LIN {X 0.113,Y -541.801,Z 1483.606,A 0.000,B 0.000,C 90.000,E1 144.975} C_DIS
LIN {X 0.190,Y -543.941,Z 1483.601,A 0.000,B 0.000,C 90.000,E1 144.116} C_DIS
LIN {X -0.031,Y -545.794,Z 1483.596,A 0.000,B 0.000,C 90.000,E1 143.290} C_DIS
LIN {X 0.087,Y -547.494,Z 1483.591,A 0.000,B 0.000,C 90.000,E1 142.431} C_DIS
LIN {X -0.159,Y -549.493,Z 1483.585,A 0.000,B 0.000,C 90.000,E1 141.331} C_DIS
LIN {X -0.082,Y -550.826,Z 1483.580,A 0.000,B 0.000,C 90.000,E1 140.481} C_DIS
LIN {X -0.278,Y -552.385,Z 1483.574,A 0.000,B 0.000,C 90.000,E1 139.380} C_DIS
LIN {X -0.042,Y -554.152,Z 1483.566,A 0.000,B 0.000,C 90.000,E1 137.957} C_DIS
LIN {X 0.124,Y -555.386,Z 1483.560,A 0.000,B 0.000,C 90.000,E1 136.824} C_DIS
LIN {X -0.011,Y -556.776,Z 1483.552,A 0.000,B 0.000,C 90.000,E1 135.445} C_DIS
LIN {X -0.192,Y -557.702,Z 1483.546,A 0.000,B 0.000,C 90.000,E1 134.352} C_DIS
LIN {X -0.236,Y -558.934,Z 1483.537,A 0.000,B 0.000,C 90.000,E1 132.690} C_DIS
LIN {X 0.038,Y -559.548,Z 1483.531,A 0.000,B 0.000,C 90.000,E1 131.553} C_DIS
LIN {X -0.100,Y -559.973,Z 1483.525,A 0.000,B 0.000,C 90.000,E1 130.458} C_DIS
LIN {X -0.079,Y -560.380,Z 1483.517,A 0.000,B 0.000,C 90.000,E1 129.072} C_DIS
LIN {X -0.139,Y -560.620,Z 1483.511,A 0.000,B 0.000,C 90.000,E1 127.971} C_DIS
LIN {X 0.086,Y -560.790,Z 1483.500,A 0.000,B 0.000,C 90.000,E1 126.011} C_DIS
LIN {X 0.236,Y -560.719,Z 1483.492,A 0.000,B 0.000,C 90.000,E1 124.612} C_DIS
LIN {X 0.120,Y -560.448,Z 1483.479,A 0.000,B 0.000,C 90.000,E1 122.133} C_DIS
LIN {X -0.123,Y -560.638,Z 1483.465,A 0.000,B 0.000,C 90.000,E1 119.667} C_DIS
LIN {X -0.105,Y -560.801,Z 1483.457,A 0.000,B 0.000,C 90.000,E1 118.281} C_DIS
LIN {X -0.254,Y -561.104,Z 1483.446,A 0.000,B 0.000,C 90.000,E1 116.360} C_DIS
LIN {X 0.113,Y -561.555,Z 1483.436,A 0.000,B 0.000,C 90.000,E1 114.387} C_DIS
LIN {X -0.087,Y -561.949,Z 1483.428,A 0.000,B 0.000,C 90.000,E1 113.025} C_DIS
LIN {X 0.050,Y -562.381,Z 1483.419,A 0.000,B 0.000,C 90.000,E1 111.354} C_DIS
LIN {X -0.136,Y -562.769,Z 1483.411,A 0.000,B 0.000,C 90.000,E1 109.993} C_DIS
LIN {X 0.014,Y -563.133,Z 1483.403,A 0.000,B 0.000,C 90.000,E1 108.598} C_DIS
LIN {X 0.310,Y -563.530,Z 1483.394,A 0.000,B 0.000,C 90.000,E1 106.913} C_DIS
LIN {X 0.145,Y -563.929,Z 1483.386,A 0.000,B 0.000,C 90.000,E1 105.552} C_DIS
LIN {X -0.090,Y -564.549,Z 1483.376,A 0.000,B 0.000,C 90.000,E1 103.647} C_DIS
LIN {X 0.020,Y -565.015,Z 1483.370,A 0.000,B 0.000,C 90.000,E1 102.535} C_DIS
LIN {X -0.077,Y -565.623,Z 1483.360,A 0.000,B 0.000,C 90.000,E1 100.894} C_DIS
LIN {X -0.271,Y -566.373,Z 1483.351,A 0.000,B 0.000,C 90.000,E1 99.265} C_DIS
LIN {X 0.194,Y -567.231,Z 1483.341,A 0.000,B 0.000,C 90.000,E1 97.296} C_DIS
LIN {X 0.039,Y -568.297,Z 1483.330,A 0.000,B 0.000,C 90.000,E1 95.391} C_DIS
LIN {X -0.192,Y -569.521,Z 1483.319,A 0.000,B 0.000,C 90.000,E1 93.498} C_DIS
LIN {X -0.100,Y -570.416,Z 1483.312,A 0.000,B 0.000,C 90.000,E1 92.121} C_DIS
LIN {X 0.139,Y -571.623,Z 1483.303,A 0.000,B 0.000,C 90.000,E1 90.458} C_DIS
LIN {X 0.096,Y -573.230,Z 1483.291,A 0.000,B 0.000,C 90.000,E1 88.282} C_DIS
LIN {X -0.156,Y -574.365,Z 1483.281,A 0.000,B 0.000,C 90.000,E1 86.674} C_DIS
LIN {X -0.233,Y -575.774,Z 1483.271,A 0.000,B 0.000,C 90.000,E1 84.780} C_DIS
LIN {X 0.197,Y -577.016,Z 1483.262,A 0.000,B 0.000,C 90.000,E1 83.109} C_DIS
LIN {X 0.153,Y -578.302,Z 1483.253,A 0.000,B 0.000,C 90.000,E1 81.489} C_DIS
LIN {X 0.232,Y -579.653,Z 1483.244,A 0.000,B 0.000,C 90.000,E1 79.859} C_DIS
LIN {X -0.230,Y -580.999,Z 1483.235,A 0.000,B 0.000,C 90.000,E1 78.285} C_DIS
LIN {X 0.122,Y -581.962,Z 1483.229,A 0.000,B 0.000,C 90.000,E1 77.173} C_DIS
LIN {X -0.044,Y -583.179,Z 1483.220,A 0.000,B 0.000,C 90.000,E1 75.574} C_DIS
LIN {X 0.148,Y -584.105,Z 1483.212,A 0.000,B 0.000,C 90.000,E1 74.212} C_DIS
LIN {X -0.217,Y -584.893,Z 1483.205,A 0.000,B 0.000,C 90.000,E1 72.906} C_DIS
LIN {X 0.005,Y -585.755,Z 1483.196,A 0.000,B 0.000,C 90.000,E1 71.275} C_DIS
LIN {X 0.027,Y -586.436,Z 1483.189,A 0.000,B 0.000,C 90.000,E1 69.934} C_DIS
LIN {X 0.060,Y -587.171,Z 1483.181,A 0.000,B 0.000,C 90.000,E1 68.592} C_DIS
LIN {X 0.159,Y -588.653,Z 1483.168,A 0.000,B 0.000,C 90.000,E1 66.177} C_DIS
LIN {X -0.177,Y -589.158,Z 1483.163,A 0.000,B 0.000,C 90.000,E1 65.409} C_DIS
LIN {X 0.136,Y -590.165,Z 1483.153,A 0.000,B 0.000,C 90.000,E1 63.512} C_DIS
LIN {X 0.102,Y -591.682,Z 1483.141,A 0.000,B 0.000,C 90.000,E1 61.385} C_DIS
LIN {X 0.071,Y -592.910,Z 1483.132,A 0.000,B 0.000,C 90.000,E1 59.793} C_DIS
LIN {X -0.038,Y -594.394,Z 1483.122,A 0.000,B 0.000,C 90.000,E1 57.946} C_DIS
LIN {X -0.325,Y -595.276,Z 1483.116,A 0.000,B 0.000,C 90.000,E1 56.914} C_DIS
LIN {X -0.143,Y -596.583,Z 1483.107,A 0.000,B 0.000,C 90.000,E1 55.308} C_DIS
LIN {X 0.069,Y -597.764,Z 1483.098,A 0.000,B 0.000,C 90.000,E1 53.703} C_DIS
LIN {X -0.063,Y -598.634,Z 1483.091,A 0.000,B 0.000,C 90.000,E1 52.396} C_DIS
LIN {X -0.178,Y -599.244,Z 1483.084,A 0.000,B 0.000,C 90.000,E1 51.090} C_DIS
LIN {X 0.094,Y -599.916,Z 1483.076,A 0.000,B 0.000,C 90.000,E1 49.747} C_DIS
LIN {X 0.114,Y -600.179,Z 1483.073,A 0.000,B 0.000,C 90.000,E1 49.218} C_DIS
LIN {X 0.158,Y -600.394,Z 1483.068,A 0.000,B 0.000,C 90.000,E1 48.162} C_DIS
LIN {X -0.017,Y -600.455,Z 1483.060,A 0.000,B 0.000,C 90.000,E1 46.863} C_DIS
LIN {X 0.202,Y -600.413,Z 1483.056,A 0.000,B 0.000,C 90.000,E1 46.053} C_DIS
LIN {X 0.007,Y -600.117,Z 1483.049,A 0.000,B 0.000,C 90.000,E1 44.757} C_DIS
LIN {X 0.225,Y -599.782,Z 1483.044,A 0.000,B 0.000,C 90.000,E1 43.947} C_DIS
LIN {X -0.401,Y -598.890,Z 1483.037,A 0.000,B 0.000,C 90.000,E1 42.690} C_DIS
LIN {X 0.246,Y -597.651,Z 1483.030,A 0.000,B 0.000,C 90.000,E1 41.310} C_DIS
LIN {X 0.254,Y -596.494,Z 1483.024,A 0.000,B 0.000,C 90.000,E1 40.253} C_DIS
LIN {X 0.019,Y -595.474,Z 1483.019,A 0.000,B 0.000,C 90.000,E1 39.483} C_DIS
LIN {X -0.165,Y -593.500,Z 1483.012,A 0.000,B 0.000,C 90.000,E1 38.177} C_DIS
LIN {X 0.096,Y -591.141,Z 1483.005,A 0.000,B 0.000,C 90.000,E1 36.824} C_DIS
LIN {X -0.365,Y -588.888,Z 1482.999,A 0.000,B 0.000,C 90.000,E1 35.804} C_DIS
LIN {X -0.101,Y -586.984,Z 1482.994,A 0.000,B 0.000,C 90.000,E1 34.978} C_DIS
LIN {X -0.339,Y -584.811,Z 1482.990,A 0.000,B 0.000,C 90.000,E1 34.199} C_DIS
LIN {X 0.028,Y -583.207,Z 1482.987,A 0.000,B 0.000,C 90.000,E1 33.627} C_DIS
LIN {X 0.058,Y -581.442,Z 1482.984,A 0.000,B 0.000,C 90.000,E1 33.086} C_DIS
LIN {X 0.084,Y -577.555,Z 1482.978,A 0.000,B 0.000,C 90.000,E1 32.005} C_DIS
LIN {X 0.078,Y -575.345,Z 1482.975,A 0.000,B 0.000,C 90.000,E1 31.465} C_DIS
LIN {X -0.110,Y -571.657,Z 1482.970,A 0.000,B 0.000,C 90.000,E1 30.669} C_DIS
LIN {X -0.249,Y -568.337,Z 1482.967,A 0.000,B 0.000,C 90.000,E1 30.001} C_DIS
LIN {X -0.111,Y -563.299,Z 1482.961,A 0.000,B 0.000,C 90.000,E1 29.027} C_DIS
LIN {X 0.167,Y -559.372,Z 1482.957,A 0.000,B 0.000,C 90.000,E1 28.309} C_DIS
LIN {X -0.086,Y -554.990,Z 1482.954,A 0.000,B 0.000,C 90.000,E1 27.641} C_DIS
LIN {X 0.081,Y -551.973,Z 1482.951,A 0.000,B 0.000,C 90.000,E1 27.206} C_DIS
LIN {X -0.007,Y -548.380,Z 1482.949,A 0.000,B 0.000,C 90.000,E1 26.796} C_DIS
LIN {X 0.252,Y -545.487,Z 1482.947,A 0.000,B 0.000,C 90.000,E1 26.488} C_DIS
LIN {X 0.255,Y -543.930,Z 1482.947,A 0.000,B 0.000,C 90.000,E1 26.360} C_DIS
LIN {X -0.225,Y -541.263,Z 1482.946,A 0.000,B 0.000,C 90.000,E1 26.232} C_DIS
LIN {X 0.063,Y -538.976,Z 1482.945,A 0.000,B 0.000,C 90.000,E1 26.104} C_DIS
LIN {X -0.136,Y -537.794,Z 1482.945,A 0.000,B 0.000,C 90.000,E1 26.104} C_DIS
LIN {X -0.121,Y -384.370,Z 1482.945,A 0.000,B 0.000,C 90.000,E1 26.104} C_DIS
LIN {X 0.078,Y -383.033,Z 1482.939,A 0.000,B 0.000,C 90.000,E1 24.951} C_DIS
LIN {X -0.114,Y -381.912,Z 1482.935,A 0.000,B 0.000,C 90.000,E1 24.259} C_DIS
LIN {X 0.134,Y -375.526,Z 1482.909,A 0.000,B 0.000,C 90.000,E1 19.504} C_DIS
LIN {X 0.003,Y -373.426,Z 1482.896,A 0.000,B 0.000,C 90.000,E1 17.330} C_DIS
LIN {X 0.014,Y -367.903,Z 1482.868,A 0.000,B 0.000,C 90.000,E1 12.175} C_DIS
LIN {X -0.043,Y -366.502,Z 1482.855,A 0.000,B 0.000,C 90.000,E1 9.962} C_DIS
LIN {X -0.108,Y -361.802,Z 1482.822,A 0.000,B 0.000,C 90.000,E1 4.012} C_DIS
LIN {X 0.138,Y -360.903,Z 1482.801,A 0.000,B 0.000,C 90.000,E1 0.229} C_DIS
LIN {X -0.053,Y -359.426,Z 1482.770,A 0.000,B 0.000,C 90.000,E1 354.546} C_DIS
LIN {X 0.070,Y -358.890,Z 1482.759,A 0.000,B 0.000,C 90.000,E1 352.648} C_DIS
LIN {X -0.020,Y -359.563,Z 1482.726,A 0.000,B 0.000,C 90.000,E1 346.645} C_DIS
LIN {X 0.001,Y -361.801,Z 1482.684,A 0.000,B 0.000,C 90.000,E1 339.135} C_DIS
LIN {X -0.154,Y -362.053,Z 1482.680,A 0.000,B 0.000,C 90.000,E1 338.411} C_DIS
LIN {X 0.189,Y -365.980,Z 1482.643,A 0.000,B 0.000,C 90.000,E1 331.641} C_DIS
LIN {X 0.029,Y -366.387,Z 1482.639,A 0.000,B 0.000,C 90.000,E1 330.923} C_DIS
LIN {X -0.031,Y -371.355,Z 1482.604,A 0.000,B 0.000,C 90.000,E1 324.642} C_DIS
LIN {X -0.043,Y -371.766,Z 1482.602,A 0.000,B 0.000,C 90.000,E1 324.276} C_DIS
LIN {X 0.013,Y -377.358,Z 1482.567,A 0.000,B 0.000,C 90.000,E1 318.038} C_DIS
LIN {X 0.012,Y -378.235,Z 1482.563,A 0.000,B 0.000,C 90.000,E1 317.310} C_DIS
LIN {X 0.002,Y -383.940,Z 1482.531,A 0.000,B 0.000,C 90.000,E1 311.515} C_DIS
LIN {X 0.088,Y -384.893,Z 1482.527,A 0.000,B 0.000,C 90.000,E1 310.782} C_DIS
LIN {X 0.262,Y -390.610,Z 1482.495,A 0.000,B 0.000,C 90.000,E1 305.025} C_DIS
LIN {X 0.106,Y -391.104,Z 1482.493,A 0.000,B 0.000,C 90.000,E1 304.692} C_DIS
LIN {X 0.022,Y -391.648,Z 1482.489,A 0.000,B 0.000,C 90.000,E1 303.992} C_DIS
LIN {X -0.080,Y -396.825,Z 1482.459,A 0.000,B 0.000,C 90.000,E1 298.693} C_DIS
LIN {X -0.210,Y -397.120,Z 1482.457,A 0.000,B 0.000,C 90.000,E1 298.359} C_DIS
LIN {X -0.055,Y -401.597,Z 1482.426,A 0.000,B 0.000,C 90.000,E1 292.717} C_DIS
LIN {X 0.222,Y -404.659,Z 1482.395,A 0.000,B 0.000,C 90.000,E1 287.094} C_DIS
LIN {X -0.079,Y -404.735,Z 1482.391,A 0.000,B 0.000,C 90.000,E1 286.441} C_DIS
LIN {X 0.214,Y -406.099,Z 1482.364,A 0.000,B 0.000,C 90.000,E1 281.535} C_DIS
LIN {X -0.176,Y -406.094,Z 1482.362,A 0.000,B 0.000,C 90.000,E1 281.243} C_DIS
LIN {X -0.097,Y -405.680,Z 1482.333,A 0.000,B 0.000,C 90.000,E1 276.024} C_DIS
LIN {X -0.165,Y -405.058,Z 1482.328,A 0.000,B 0.000,C 90.000,E1 274.992} C_DIS
LIN {X -0.060,Y -403.497,Z 1482.304,A 0.000,B 0.000,C 90.000,E1 270.802} C_DIS
LIN {X -0.092,Y -403.288,Z 1482.302,A 0.000,B 0.000,C 90.000,E1 270.458} C_DIS
LIN {X 0.091,Y -398.931,Z 1482.271,A 0.000,B 0.000,C 90.000,E1 264.837} C_DIS
LIN {X -0.040,Y -393.108,Z 1482.242,A 0.000,B 0.000,C 90.000,E1 259.567} C_DIS
LIN {X -0.079,Y -392.835,Z 1482.240,A 0.000,B 0.000,C 90.000,E1 259.218} C_DIS
LIN {X 0.034,Y -385.993,Z 1482.212,A 0.000,B 0.000,C 90.000,E1 254.212} C_DIS
LIN {X -0.026,Y -385.267,Z 1482.208,A 0.000,B 0.000,C 90.000,E1 253.504} C_DIS
LIN {X -0.004,Y -384.768,Z 1482.206,A 0.000,B 0.000,C 90.000,E1 253.142} C_DIS
LIN {X 0.221,Y -377.973,Z 1482.182,A 0.000,B 0.000,C 90.000,E1 248.773} C_DIS
LIN {X -0.044,Y -376.233,Z 1482.174,A 0.000,B 0.000,C 90.000,E1 247.358} C_DIS
LIN {X 0.057,Y -374.944,Z 1482.170,A 0.000,B 0.000,C 90.000,E1 246.613} C_DIS
LIN {X -0.208,Y -368.417,Z 1482.148,A 0.000,B 0.000,C 90.000,E1 242.615} C_DIS
LIN {X 0.097,Y -366.047,Z 1482.137,A 0.000,B 0.000,C 90.000,E1 240.717} C_DIS
LIN {X 0.004,Y -359.196,Z 1482.115,A 0.000,B 0.000,C 90.000,E1 236.628} C_DIS
LIN {X 0.021,Y -355.842,Z 1482.100,A 0.000,B 0.000,C 90.000,E1 233.989} C_DIS
LIN {X -0.173,Y -348.793,Z 1482.075,A 0.000,B 0.000,C 90.000,E1 229.461} C_DIS
LIN {X -0.097,Y -346.185,Z 1482.062,A 0.000,B 0.000,C 90.000,E1 227.148} C_DIS
LIN {X -0.088,Y -345.065,Z 1482.058,A 0.000,B 0.000,C 90.000,E1 226.377} C_DIS
LIN {X 0.094,Y -338.586,Z 1482.030,A 0.000,B 0.000,C 90.000,E1 221.310} C_DIS
LIN {X 0.094,Y -336.840,Z 1482.019,A 0.000,B 0.000,C 90.000,E1 219.358} C_DIS
LIN {X 0.014,Y -330.861,Z 1481.988,A 0.000,B 0.000,C 90.000,E1 213.865} C_DIS
LIN {X 0.149,Y -329.296,Z 1481.975,A 0.000,B 0.000,C 90.000,E1 211.465} C_DIS
LIN {X -0.154,Y -324.669,Z 1481.942,A 0.000,B 0.000,C 90.000,E1 205.540} C_DIS
LIN {X 0.174,Y -323.837,Z 1481.928,A 0.000,B 0.000,C 90.000,E1 203.078} C_DIS
LIN {X -0.017,Y -321.124,Z 1481.881,A 0.000,B 0.000,C 90.000,E1 194.662} C_DIS
LIN {X 0.138,Y -320.932,Z 1481.877,A 0.000,B 0.000,C 90.000,E1 193.828} C_DIS
LIN {X -0.076,Y -321.562,Z 1481.832,A 0.000,B 0.000,C 90.000,E1 185.796} C_DIS
LIN {X -0.143,Y -324.415,Z 1481.790,A 0.000,B 0.000,C 90.000,E1 178.165} C_DIS
LIN {X -0.141,Y -325.376,Z 1481.783,A 0.000,B 0.000,C 90.000,E1 176.963} C_DIS
LIN {X -0.100,Y -329.112,Z 1481.750,A 0.000,B 0.000,C 90.000,E1 170.971} C_DIS
LIN {X 0.061,Y -334.260,Z 1481.726,A 0.000,B 0.000,C 90.000,E1 166.589} C_DIS
LIN {X 0.067,Y -335.488,Z 1481.719,A 0.000,B 0.000,C 90.000,E1 165.408} C_DIS
LIN {X 0.143,Y -340.932,Z 1481.695,A 0.000,B 0.000,C 90.000,E1 161.094} C_DIS
LIN {X -0.172,Y -342.138,Z 1481.691,A 0.000,B 0.000,C 90.000,E1 160.369} C_DIS
LIN {X -0.058,Y -347.939,Z 1481.667,A 0.000,B 0.000,C 90.000,E1 156.102} C_DIS
LIN {X 0.037,Y -354.622,Z 1481.647,A 0.000,B 0.000,C 90.000,E1 152.436} C_DIS
LIN {X 0.000,Y -354.671,Z 1481.647,A 0.000,B 0.000,C 90.000,E1 152.410} C_DIS
LIN {X -0.047,Y -501.646,Z 1481.647,A 0.000,B 0.000,C 90.000,E1 152.410} C_DIS
LIN {X -0.075,Y -505.220,Z 1481.646,A 0.000,B 0.000,C 90.000,E1 152.281} C_DIS
LIN {X -0.137,Y -507.377,Z 1481.645,A 0.000,B 0.000,C 90.000,E1 152.153} C_DIS
LIN {X -0.108,Y -509.939,Z 1481.644,A 0.000,B 0.000,C 90.000,E1 151.948} C_DIS
LIN {X -0.018,Y -513.664,Z 1481.642,A 0.000,B 0.000,C 90.000,E1 151.563} C_DIS
LIN {X 0.194,Y -515.980,Z 1481.641,A 0.000,B 0.000,C 90.000,E1 151.257} C_DIS
LIN {X -0.069,Y -519.084,Z 1481.638,A 0.000,B 0.000,C 90.000,E1 150.845} C_DIS
LIN {X -0.026,Y -522.481,Z 1481.635,A 0.000,B 0.000,C 90.000,E1 150.255} C_DIS
LIN {X -0.117,Y -526.265,Z 1481.631,A 0.000,B 0.000,C 90.000,E1 149.537} C_DIS
LIN {X 0.091,Y -529.473,Z 1481.627,A 0.000,B 0.000,C 90.000,E1 148.791} C_DIS
LIN {X 0.207,Y -531.888,Z 1481.624,A 0.000,B 0.000,C 90.000,E1 148.201} C_DIS
LIN {X -0.117,Y -534.035,Z 1481.620,A 0.000,B 0.000,C 90.000,E1 147.661} C_DIS
LIN {X 0.013,Y -536.921,Z 1481.615,A 0.000,B 0.000,C 90.000,E1 146.786} C_DIS
LIN {X 0.026,Y -539.502,Z 1481.611,A 0.000,B 0.000,C 90.000,E1 145.928} C_DIS
LIN {X -0.232,Y -541.972,Z 1481.606,A 0.000,B 0.000,C 90.000,E1 145.102} C_DIS
LIN {X 0.289,Y -544.154,Z 1481.601,A 0.000,B 0.000,C 90.000,E1 144.196} C_DIS
LIN {X 0.069,Y -546.018,Z 1481.597,A 0.000,B 0.000,C 90.000,E1 143.371} C_DIS
LIN {X -0.201,Y -548.230,Z 1481.590,A 0.000,B 0.000,C 90.000,E1 142.271} C_DIS
LIN {X -0.056,Y -549.722,Z 1481.586,A 0.000,B 0.000,C 90.000,E1 141.412} C_DIS
LIN {X 0.078,Y -551.419,Z 1481.579,A 0.000,B 0.000,C 90.000,E1 140.275} C_DIS
LIN {X -0.116,Y -552.960,Z 1481.573,A 0.000,B 0.000,C 90.000,E1 139.175} C_DIS
LIN {X 0.067,Y -554.326,Z 1481.567,A 0.000,B 0.000,C 90.000,E1 138.038} C_DIS
LIN {X -0.111,Y -555.828,Z 1481.559,A 0.000,B 0.000,C 90.000,E1 136.662} C_DIS
LIN {X 0.152,Y -557.194,Z 1481.552,A 0.000,B 0.000,C 90.000,E1 135.243} C_DIS
LIN {X 0.035,Y -558.250,Z 1481.544,A 0.000,B 0.000,C 90.000,E1 133.866} C_DIS
LIN {X -0.041,Y -559.241,Z 1481.536,A 0.000,B 0.000,C 90.000,E1 132.486} C_DIS
LIN {X -0.176,Y -559.800,Z 1481.530,A 0.000,B 0.000,C 90.000,E1 131.391} C_DIS
LIN {X -0.226,Y -560.240,Z 1481.522,A 0.000,B 0.000,C 90.000,E1 130.011} C_DIS
LIN {X -0.199,Y -560.596,Z 1481.515,A 0.000,B 0.000,C 90.000,E1 128.624} C_DIS
LIN {X -0.163,Y -560.744,Z 1481.507,A 0.000,B 0.000,C 90.000,E1 127.237} C_DIS
LIN {X 0.318,Y -560.835,Z 1481.499,A 0.000,B 0.000,C 90.000,E1 125.804} C_DIS
LIN {X -0.084,Y -560.757,Z 1481.493,A 0.000,B 0.000,C 90.000,E1 124.739} C_DIS
LIN {X 0.057,Y -560.447,Z 1481.478,A 0.000,B 0.000,C 90.000,E1 121.957} C_DIS
LIN {X 0.033,Y -560.619,Z 1481.465,A 0.000,B 0.000,C 90.000,E1 119.745} C_DIS
LIN {X -0.146,Y -560.817,Z 1481.456,A 0.000,B 0.000,C 90.000,E1 118.103} C_DIS
LIN {X -0.086,Y -561.090,Z 1481.447,A 0.000,B 0.000,C 90.000,E1 116.437} C_DIS
LIN {X -0.221,Y -561.538,Z 1481.436,A 0.000,B 0.000,C 90.000,E1 114.515} C_DIS
LIN {X 0.116,Y -562.010,Z 1481.427,A 0.000,B 0.000,C 90.000,E1 112.823} C_DIS
LIN {X 0.038,Y -562.486,Z 1481.418,A 0.000,B 0.000,C 90.000,E1 111.173} C_DIS
LIN {X -0.145,Y -562.844,Z 1481.410,A 0.000,B 0.000,C 90.000,E1 109.812} C_DIS
LIN {X 0.147,Y -563.278,Z 1481.401,A 0.000,B 0.000,C 90.000,E1 108.127} C_DIS
LIN {X 0.064,Y -563.801,Z 1481.390,A 0.000,B 0.000,C 90.000,E1 106.205} C_DIS
LIN {X 0.215,Y -564.288,Z 1481.381,A 0.000,B 0.000,C 90.000,E1 104.537} C_DIS
LIN {X -0.156,Y -565.017,Z 1481.370,A 0.000,B 0.000,C 90.000,E1 102.647} C_DIS
LIN {X 0.296,Y -565.653,Z 1481.361,A 0.000,B 0.000,C 90.000,E1 100.950} C_DIS
LIN {X -0.207,Y -566.629,Z 1481.349,A 0.000,B 0.000,C 90.000,E1 98.803} C_DIS
LIN {X -0.196,Y -567.682,Z 1481.337,A 0.000,B 0.000,C 90.000,E1 96.606} C_DIS
LIN {X 0.066,Y -568.632,Z 1481.328,A 0.000,B 0.000,C 90.000,E1 94.935} C_DIS
LIN {X -0.114,Y -569.903,Z 1481.317,A 0.000,B 0.000,C 90.000,E1 93.037} C_DIS
LIN {X 0.107,Y -571.045,Z 1481.308,A 0.000,B 0.000,C 90.000,E1 91.375} C_DIS
LIN {X 0.208,Y -572.009,Z 1481.300,A 0.000,B 0.000,C 90.000,E1 90.000} C_DIS
LIN {X -0.106,Y -573.258,Z 1481.291,A 0.000,B 0.000,C 90.000,E1 88.396} C_DIS
LIN {X 0.217,Y -574.426,Z 1481.282,A 0.000,B 0.000,C 90.000,E1 86.731} C_DIS
LIN {X 0.144,Y -575.851,Z 1481.271,A 0.000,B 0.000,C 90.000,E1 84.837} C_DIS
LIN {X 0.005,Y -577.111,Z 1481.262,A 0.000,B 0.000,C 90.000,E1 83.223} C_DIS
LIN {X -0.247,Y -578.199,Z 1481.255,A 0.000,B 0.000,C 90.000,E1 81.894} C_DIS
LIN {X -0.270,Y -579.539,Z 1481.246,A 0.000,B 0.000,C 90.000,E1 80.274} C_DIS
LIN {X -0.061,Y -580.925,Z 1481.237,A 0.000,B 0.000,C 90.000,E1 78.634} C_DIS
LIN {X 0.190,Y -582.338,Z 1481.228,A 0.000,B 0.000,C 90.000,E1 76.992} C_DIS
LIN {X -0.110,Y -583.542,Z 1481.219,A 0.000,B 0.000,C 90.000,E1 75.408} C_DIS
LIN {X 0.076,Y -584.419,Z 1481.211,A 0.000,B 0.000,C 90.000,E1 74.047} C_DIS
LIN {X -0.121,Y -585.200,Z 1481.204,A 0.000,B 0.000,C 90.000,E1 72.725} C_DIS
LIN {X -0.225,Y -586.253,Z 1481.194,A 0.000,B 0.000,C 90.000,E1 70.859} C_DIS
LIN {X -0.249,Y -587.353,Z 1481.182,A 0.000,B 0.000,C 90.000,E1 68.720} C_DIS
LIN {X 0.315,Y -588.454,Z 1481.171,A 0.000,B 0.000,C 90.000,E1 66.794} C_DIS
LIN {X 0.050,Y -589.326,Z 1481.164,A 0.000,B 0.000,C 90.000,E1 65.485} C_DIS
LIN {X -0.170,Y -590.341,Z 1481.154,A 0.000,B 0.000,C 90.000,E1 63.640} C_DIS
LIN {X -0.096,Y -591.604,Z 1481.143,A 0.000,B 0.000,C 90.000,E1 61.769} C_DIS
LIN {X -0.319,Y -592.662,Z 1481.136,A 0.000,B 0.000,C 90.000,E1 60.461} C_DIS
LIN {X -0.224,Y -594.346,Z 1481.124,A 0.000,B 0.000,C 90.000,E1 58.329} C_DIS
LIN {X -0.111,Y -595.444,Z 1481.117,A 0.000,B 0.000,C 90.000,E1 56.993} C_DIS
LIN {X 0.070,Y -596.770,Z 1481.108,A 0.000,B 0.000,C 90.000,E1 55.388} C_DIS
LIN {X -0.200,Y -597.960,Z 1481.099,A 0.000,B 0.000,C 90.000,E1 53.829} C_DIS
LIN {X 0.151,Y -598.865,Z 1481.092,A 0.000,B 0.000,C 90.000,E1 52.477} C_DIS
LIN {X 0.038,Y -599.514,Z 1481.084,A 0.000,B 0.000,C 90.000,E1 51.170} C_DIS
LIN {X 0.312,Y -600.176,Z 1481.077,A 0.000,B 0.000,C 90.000,E1 49.828} C_DIS
LIN {X 0.119,Y -600.525,Z 1481.073,A 0.000,B 0.000,C 90.000,E1 49.057} C_DIS
LIN {X 0.381,Y -600.692,Z 1481.068,A 0.000,B 0.000,C 90.000,E1 48.243} C_DIS
LIN {X -0.228,Y -600.762,Z 1481.061,A 0.000,B 0.000,C 90.000,E1 46.986} C_DIS
LIN {X -0.001,Y -600.734,Z 1481.057,A 0.000,B 0.000,C 90.000,E1 46.176} C_DIS
LIN {X 0.241,Y -600.466,Z 1481.049,A 0.000,B 0.000,C 90.000,E1 44.838} C_DIS
LIN {X 0.254,Y -599.989,Z 1481.043,A 0.000,B 0.000,C 90.000,E1 43.785} C_DIS
LIN {X 0.072,Y -599.083,Z 1481.036,A 0.000,B 0.000,C 90.000,E1 42.486} C_DIS
LIN {X 0.051,Y -598.104,Z 1481.030,A 0.000,B 0.000,C 90.000,E1 41.434} C_DIS
LIN {X 0.059,Y -596.947,Z 1481.024,A 0.000,B 0.000,C 90.000,E1 40.378} C_DIS
LIN {X 0.050,Y -595.527,Z 1481.019,A 0.000,B 0.000,C 90.000,E1 39.322} C_DIS
LIN {X 0.110,Y -593.991,Z 1481.013,A 0.000,B 0.000,C 90.000,E1 38.257} C_DIS
LIN {X -0.093,Y -591.687,Z 1481.005,A 0.000,B 0.000,C 90.000,E1 36.950} C_DIS
LIN {X -0.073,Y -589.493,Z 1480.999,A 0.000,B 0.000,C 90.000,E1 35.884} C_DIS
LIN {X -0.283,Y -587.620,Z 1480.995,A 0.000,B 0.000,C 90.000,E1 35.105} C_DIS
LIN {X -0.030,Y -585.505,Z 1480.990,A 0.000,B 0.000,C 90.000,E1 34.278} C_DIS
LIN {X -0.286,Y -583.094,Z 1480.986,A 0.000,B 0.000,C 90.000,E1 33.499} C_DIS
LIN {X -0.234,Y -579.480,Z 1480.980,A 0.000,B 0.000,C 90.000,E1 32.418} C_DIS
LIN {X -0.225,Y -577.441,Z 1480.977,A 0.000,B 0.000,C 90.000,E1 31.878} C_DIS
LIN {X -0.090,Y -573.965,Z 1480.973,A 0.000,B 0.000,C 90.000,E1 31.052} C_DIS
LIN {X 0.114,Y -569.519,Z 1480.967,A 0.000,B 0.000,C 90.000,E1 30.079} C_DIS
LIN {X -0.141,Y -563.024,Z 1480.960,A 0.000,B 0.000,C 90.000,E1 28.871} C_DIS
LIN {X -0.035,Y -559.907,Z 1480.957,A 0.000,B 0.000,C 90.000,E1 28.309} C_DIS
LIN {X 0.209,Y -555.559,Z 1480.953,A 0.000,B 0.000,C 90.000,E1 27.590} C_DIS
LIN {X 0.030,Y -551.830,Z 1480.950,A 0.000,B 0.000,C 90.000,E1 27.052} C_DIS
LIN {X 0.182,Y -548.690,Z 1480.948,A 0.000,B 0.000,C 90.000,E1 26.616} C_DIS
LIN {X -0.173,Y -544.957,Z 1480.946,A 0.000,B 0.000,C 90.000,E1 26.232} C_DIS
LIN {X 0.146,Y -542.086,Z 1480.944,A 0.000,B 0.000,C 90.000,E1 25.924} C_DIS
LIN {X 0.096,Y -540.475,Z 1480.943,A 0.000,B 0.000,C 90.000,E1 25.796} C_DIS
LIN {X 0.170,Y -538.760,Z 1480.943,A 0.000,B 0.000,C 90.000,E1 25.668} C_DIS
LIN {X 0.035,Y -535.864,Z 1480.942,A 0.000,B 0.000,C 90.000,E1 25.540} C_DIS
LIN {X -0.035,Y -534.505,Z 1480.942,A 0.000,B 0.000,C 90.000,E1 25.515} C_DIS
LIN {X -0.054,Y -383.662,Z 1480.942,A 0.000,B 0.000,C 90.000,E1 25.515} C_DIS
LIN {X 0.191,Y -382.637,Z 1480.937,A 0.000,B 0.000,C 90.000,E1 24.643} C_DIS
LIN {X 0.130,Y -375.997,Z 1480.911,A 0.000,B 0.000,C 90.000,E1 19.939} C_DIS
LIN {X -0.006,Y -373.524,Z 1480.897,A 0.000,B 0.000,C 90.000,E1 17.402} C_DIS
LIN {X 0.033,Y -367.958,Z 1480.868,A 0.000,B 0.000,C 90.000,E1 12.243} C_DIS
LIN {X 0.051,Y -366.538,Z 1480.856,A 0.000,B 0.000,C 90.000,E1 10.018} C_DIS
LIN {X -0.020,Y -365.428,Z 1480.850,A 0.000,B 0.000,C 90.000,E1 8.916} C_DIS
LIN {X -0.055,Y -361.273,Z 1480.814,A 0.000,B 0.000,C 90.000,E1 2.579} C_DIS
LIN {X -0.130,Y -360.906,Z 1480.802,A 0.000,B 0.000,C 90.000,E1 0.344} C_DIS
LIN {X 0.044,Y -359.764,Z 1480.786,A 0.000,B 0.000,C 90.000,E1 357.535} C_DIS
LIN {X -0.053,Y -359.426,Z 1480.770,A 0.000,B 0.000,C 90.000,E1 354.546} C_DIS
LIN {X 0.070,Y -358.890,Z 1480.759,A 0.000,B 0.000,C 90.000,E1 352.648} C_DIS
LIN {X -0.020,Y -359.563,Z 1480.726,A 0.000,B 0.000,C 90.000,E1 346.645} C_DIS
LIN {X 0.001,Y -361.801,Z 1480.684,A 0.000,B 0.000,C 90.000,E1 339.135} C_DIS
LIN {X -0.154,Y -362.053,Z 1480.680,A 0.000,B 0.000,C 90.000,E1 338.411} C_DIS
LIN {X 0.189,Y -365.980,Z 1480.643,A 0.000,B 0.000,C 90.000,E1 331.641} C_DIS
LIN {X 0.029,Y -366.387,Z 1480.639,A 0.000,B 0.000,C 90.000,E1 330.923} C_DIS
LIN {X -0.031,Y -371.355,Z 1480.604,A 0.000,B 0.000,C 90.000,E1 324.642} C_DIS
LIN {X -0.043,Y -371.766,Z 1480.602,A 0.000,B 0.000,C 90.000,E1 324.276} C_DIS
LIN {X 0.013,Y -377.358,Z 1480.567,A 0.000,B 0.000,C 90.000,E1 318.038} C_DIS
LIN {X 0.012,Y -378.235,Z 1480.563,A 0.000,B 0.000,C 90.000,E1 317.310} C_DIS
LIN {X 0.002,Y -383.940,Z 1480.531,A 0.000,B 0.000,C 90.000,E1 311.515} C_DIS
LIN {X 0.088,Y -384.893,Z 1480.527,A 0.000,B 0.000,C 90.000,E1 310.782} C_DIS
LIN {X 0.262,Y -390.610,Z 1480.495,A 0.000,B 0.000,C 90.000,E1 305.025} C_DIS
LIN {X 0.106,Y -391.104,Z 1480.493,A 0.000,B 0.000,C 90.000,E1 304.692} C_DIS
LIN {X 0.022,Y -391.648,Z 1480.489,A 0.000,B 0.000,C 90.000,E1 303.992} C_DIS
LIN {X -0.080,Y -396.825,Z 1480.459,A 0.000,B 0.000,C 90.000,E1 298.693} C_DIS
LIN {X -0.210,Y -397.120,Z 1480.457,A 0.000,B 0.000,C 90.000,E1 298.359} C_DIS
LIN {X -0.055,Y -401.597,Z 1480.426,A 0.000,B 0.000,C 90.000,E1 292.717} C_DIS
LIN {X 0.222,Y -404.659,Z 1480.395,A 0.000,B 0.000,C 90.000,E1 287.094} C_DIS
LIN {X -0.079,Y -404.735,Z 1480.391,A 0.000,B 0.000,C 90.000,E1 286.441} C_DIS
LIN {X 0.214,Y -406.099,Z 1480.364,A 0.000,B 0.000,C 90.000,E1 281.535} C_DIS
LIN {X -0.176,Y -406.094,Z 1480.362,A 0.000,B 0.000,C 90.000,E1 281.243} C_DIS
LIN {X -0.097,Y -405.680,Z 1480.333,A 0.000,B 0.000,C 90.000,E1 276.024} C_DIS
LIN {X -0.165,Y -405.058,Z 1480.328,A 0.000,B 0.000,C 90.000,E1 274.992} C_DIS
LIN {X -0.060,Y -403.497,Z 1480.304,A 0.000,B 0.000,C 90.000,E1 270.802} C_DIS
LIN {X -0.092,Y -403.288,Z 1480.302,A 0.000,B 0.000,C 90.000,E1 270.458} C_DIS
LIN {X 0.091,Y -398.931,Z 1480.271,A 0.000,B 0.000,C 90.000,E1 264.837} C_DIS
LIN {X -0.040,Y -393.108,Z 1480.242,A 0.000,B 0.000,C 90.000,E1 259.567} C_DIS
LIN {X -0.079,Y -392.835,Z 1480.240,A 0.000,B 0.000,C 90.000,E1 259.218} C_DIS
LIN {X 0.034,Y -385.993,Z 1480.212,A 0.000,B 0.000,C 90.000,E1 254.212} C_DIS
LIN {X -0.026,Y -385.267,Z 1480.208,A 0.000,B 0.000,C 90.000,E1 253.504} C_DIS
LIN {X -0.004,Y -384.768,Z 1480.206,A 0.000,B 0.000,C 90.000,E1 253.142} C_DIS
LIN {X 0.221,Y -377.973,Z 1480.182,A 0.000,B 0.000,C 90.000,E1 248.773} C_DIS
LIN {X -0.044,Y -376.233,Z 1480.174,A 0.000,B 0.000,C 90.000,E1 247.358} C_DIS
LIN {X 0.057,Y -374.944,Z 1480.170,A 0.000,B 0.000,C 90.000,E1 246.613} C_DIS
LIN {X -0.208,Y -368.417,Z 1480.148,A 0.000,B 0.000,C 90.000,E1 242.615} C_DIS
LIN {X 0.097,Y -366.047,Z 1480.137,A 0.000,B 0.000,C 90.000,E1 240.717} C_DIS
LIN {X 0.004,Y -359.196,Z 1480.115,A 0.000,B 0.000,C 90.000,E1 236.628} C_DIS
LIN {X 0.021,Y -355.842,Z 1480.100,A 0.000,B 0.000,C 90.000,E1 233.989} C_DIS
LIN {X -0.173,Y -348.793,Z 1480.075,A 0.000,B 0.000,C 90.000,E1 229.461} C_DIS
LIN {X -0.097,Y -346.185,Z 1480.062,A 0.000,B 0.000,C 90.000,E1 227.148} C_DIS
LIN {X -0.088,Y -345.065,Z 1480.058,A 0.000,B 0.000,C 90.000,E1 226.377} C_DIS
LIN {X 0.094,Y -338.586,Z 1480.030,A 0.000,B 0.000,C 90.000,E1 221.310} C_DIS
LIN {X 0.094,Y -336.840,Z 1480.019,A 0.000,B 0.000,C 90.000,E1 219.358} C_DIS
LIN {X 0.014,Y -330.861,Z 1479.988,A 0.000,B 0.000,C 90.000,E1 213.865} C_DIS
LIN {X 0.149,Y -329.296,Z 1479.975,A 0.000,B 0.000,C 90.000,E1 211.465} C_DIS
LIN {X -0.154,Y -324.669,Z 1479.942,A 0.000,B 0.000,C 90.000,E1 205.540} C_DIS
LIN {X 0.174,Y -323.837,Z 1479.928,A 0.000,B 0.000,C 90.000,E1 203.078} C_DIS
LIN {X -0.017,Y -321.124,Z 1479.881,A 0.000,B 0.000,C 90.000,E1 194.662} C_DIS
LIN {X 0.138,Y -320.932,Z 1479.877,A 0.000,B 0.000,C 90.000,E1 193.828} C_DIS
LIN {X -0.076,Y -321.562,Z 1479.832,A 0.000,B 0.000,C 90.000,E1 185.796} C_DIS
LIN {X -0.143,Y -324.415,Z 1479.790,A 0.000,B 0.000,C 90.000,E1 178.165} C_DIS
LIN {X -0.141,Y -325.376,Z 1479.783,A 0.000,B 0.000,C 90.000,E1 176.963} C_DIS
LIN {X -0.100,Y -329.112,Z 1479.750,A 0.000,B 0.000,C 90.000,E1 170.971} C_DIS
LIN {X 0.061,Y -334.260,Z 1479.726,A 0.000,B 0.000,C 90.000,E1 166.589} C_DIS
LIN {X 0.067,Y -335.488,Z 1479.719,A 0.000,B 0.000,C 90.000,E1 165.408} C_DIS
LIN {X 0.143,Y -340.932,Z 1479.695,A 0.000,B 0.000,C 90.000,E1 161.094} C_DIS
LIN {X -0.172,Y -342.138,Z 1479.691,A 0.000,B 0.000,C 90.000,E1 160.369} C_DIS
LIN {X -0.058,Y -347.939,Z 1479.667,A 0.000,B 0.000,C 90.000,E1 156.102} C_DIS
LIN {X -0.069,Y -353.576,Z 1479.650,A 0.000,B 0.000,C 90.000,E1 152.999} C_DIS
LIN {X -0.123,Y -497.290,Z 1479.650,A 0.000,B 0.000,C 90.000,E1 152.999} C_DIS
LIN {X -0.140,Y -500.027,Z 1479.650,A 0.000,B 0.000,C 90.000,E1 152.922} C_DIS
LIN {X 0.062,Y -501.637,Z 1479.649,A 0.000,B 0.000,C 90.000,E1 152.820} C_DIS
LIN {X -0.116,Y -504.385,Z 1479.648,A 0.000,B 0.000,C 90.000,E1 152.666} C_DIS
LIN {X 0.104,Y -506.939,Z 1479.647,A 0.000,B 0.000,C 90.000,E1 152.436} C_DIS
LIN {X -0.279,Y -510.846,Z 1479.645,A 0.000,B 0.000,C 90.000,E1 152.103} C_DIS
LIN {X -0.007,Y -514.398,Z 1479.642,A 0.000,B 0.000,C 90.000,E1 151.641} C_DIS
LIN {X 0.094,Y -516.525,Z 1479.641,A 0.000,B 0.000,C 90.000,E1 151.335} C_DIS
LIN {X 0.114,Y -520.206,Z 1479.638,A 0.000,B 0.000,C 90.000,E1 150.745} C_DIS
LIN {X 0.261,Y -524.228,Z 1479.634,A 0.000,B 0.000,C 90.000,E1 149.999} C_DIS
LIN {X 0.045,Y -526.497,Z 1479.631,A 0.000,B 0.000,C 90.000,E1 149.587} C_DIS
LIN {X -0.168,Y -530.315,Z 1479.626,A 0.000,B 0.000,C 90.000,E1 148.742} C_DIS
LIN {X 0.231,Y -532.670,Z 1479.623,A 0.000,B 0.000,C 90.000,E1 148.122} C_DIS
LIN {X -0.087,Y -534.770,Z 1479.620,A 0.000,B 0.000,C 90.000,E1 147.582} C_DIS
LIN {X 0.054,Y -537.604,Z 1479.615,A 0.000,B 0.000,C 90.000,E1 146.707} C_DIS
LIN {X 0.063,Y -539.360,Z 1479.612,A 0.000,B 0.000,C 90.000,E1 146.135} C_DIS
LIN {X 0.272,Y -542.614,Z 1479.606,A 0.000,B 0.000,C 90.000,E1 144.975} C_DIS
LIN {X 0.039,Y -544.727,Z 1479.601,A 0.000,B 0.000,C 90.000,E1 144.149} C_DIS
LIN {X 0.107,Y -546.008,Z 1479.598,A 0.000,B 0.000,C 90.000,E1 143.577} C_DIS
LIN {X -0.161,Y -548.199,Z 1479.592,A 0.000,B 0.000,C 90.000,E1 142.477} C_DIS
LIN {X 0.037,Y -550.182,Z 1479.585,A 0.000,B 0.000,C 90.000,E1 141.331} C_DIS
LIN {X 0.180,Y -551.843,Z 1479.579,A 0.000,B 0.000,C 90.000,E1 140.194} C_DIS
LIN {X -0.006,Y -553.357,Z 1479.573,A 0.000,B 0.000,C 90.000,E1 139.094} C_DIS
LIN {X 0.124,Y -554.376,Z 1479.568,A 0.000,B 0.000,C 90.000,E1 138.243} C_DIS
LIN {X -0.023,Y -555.909,Z 1479.560,A 0.000,B 0.000,C 90.000,E1 136.863} C_DIS
LIN {X -0.166,Y -557.207,Z 1479.553,A 0.000,B 0.000,C 90.000,E1 135.486} C_DIS
LIN {X -0.281,Y -558.302,Z 1479.545,A 0.000,B 0.000,C 90.000,E1 134.109} C_DIS
LIN {X 0.022,Y -559.320,Z 1479.537,A 0.000,B 0.000,C 90.000,E1 132.690} C_DIS
LIN {X -0.117,Y -559.880,Z 1479.531,A 0.000,B 0.000,C 90.000,E1 131.595} C_DIS
LIN {X 0.169,Y -560.250,Z 1479.525,A 0.000,B 0.000,C 90.000,E1 130.458} C_DIS
LIN {X -0.148,Y -560.614,Z 1479.516,A 0.000,B 0.000,C 90.000,E1 128.830} C_DIS
LIN {X -0.116,Y -560.784,Z 1479.508,A 0.000,B 0.000,C 90.000,E1 127.443} C_DIS
LIN {X 0.364,Y -560.894,Z 1479.500,A 0.000,B 0.000,C 90.000,E1 126.011} C_DIS
LIN {X -0.038,Y -560.803,Z 1479.494,A 0.000,B 0.000,C 90.000,E1 124.945} C_DIS
LIN {X -0.157,Y -560.458,Z 1479.480,A 0.000,B 0.000,C 90.000,E1 122.467} C_DIS
LIN {X -0.196,Y -560.559,Z 1479.468,A 0.000,B 0.000,C 90.000,E1 120.256} C_DIS
LIN {X -0.091,Y -560.791,Z 1479.457,A 0.000,B 0.000,C 90.000,E1 118.309} C_DIS
LIN {X 0.226,Y -561.062,Z 1479.448,A 0.000,B 0.000,C 90.000,E1 116.616} C_DIS
LIN {X -0.152,Y -561.466,Z 1479.437,A 0.000,B 0.000,C 90.000,E1 114.719} C_DIS
LIN {X 0.194,Y -562.002,Z 1479.428,A 0.000,B 0.000,C 90.000,E1 113.025} C_DIS
LIN {X 0.125,Y -562.562,Z 1479.417,A 0.000,B 0.000,C 90.000,E1 111.099} C_DIS
LIN {X -0.336,Y -563.053,Z 1479.407,A 0.000,B 0.000,C 90.000,E1 109.214} C_DIS
LIN {X -0.177,Y -563.396,Z 1479.399,A 0.000,B 0.000,C 90.000,E1 107.819} C_DIS
LIN {X 0.276,Y -563.935,Z 1479.388,A 0.000,B 0.000,C 90.000,E1 105.843} C_DIS
LIN {X 0.038,Y -564.559,Z 1479.378,A 0.000,B 0.000,C 90.000,E1 103.939} C_DIS
LIN {X 0.093,Y -565.307,Z 1479.367,A 0.000,B 0.000,C 90.000,E1 102.007} C_DIS
LIN {X -0.170,Y -565.847,Z 1479.359,A 0.000,B 0.000,C 90.000,E1 100.658} C_DIS
LIN {X -0.281,Y -566.720,Z 1479.349,A 0.000,B 0.000,C 90.000,E1 98.746} C_DIS
LIN {X -0.201,Y -567.782,Z 1479.336,A 0.000,B 0.000,C 90.000,E1 96.543} C_DIS
LIN {X 0.000,Y -568.739,Z 1479.327,A 0.000,B 0.000,C 90.000,E1 94.878} C_DIS
LIN {X -0.176,Y -570.010,Z 1479.317,A 0.000,B 0.000,C 90.000,E1 92.980} C_DIS
LIN {X 0.048,Y -571.185,Z 1479.307,A 0.000,B 0.000,C 90.000,E1 91.318} C_DIS
LIN {X -0.282,Y -572.345,Z 1479.298,A 0.000,B 0.000,C 90.000,E1 89.714} C_DIS
LIN {X -0.160,Y -573.408,Z 1479.291,A 0.000,B 0.000,C 90.000,E1 88.339} C_DIS
LIN {X 0.166,Y -574.607,Z 1479.282,A 0.000,B 0.000,C 90.000,E1 86.674} C_DIS
LIN {X 0.095,Y -576.042,Z 1479.271,A 0.000,B 0.000,C 90.000,E1 84.780} C_DIS
LIN {X -0.040,Y -577.320,Z 1479.262,A 0.000,B 0.000,C 90.000,E1 83.166} C_DIS
LIN {X -0.291,Y -578.441,Z 1479.255,A 0.000,B 0.000,C 90.000,E1 81.837} C_DIS
LIN {X 0.136,Y -579.561,Z 1479.247,A 0.000,B 0.000,C 90.000,E1 80.443} C_DIS
LIN {X -0.101,Y -581.190,Z 1479.237,A 0.000,B 0.000,C 90.000,E1 78.578} C_DIS
LIN {X 0.153,Y -582.612,Z 1479.228,A 0.000,B 0.000,C 90.000,E1 76.937} C_DIS
LIN {X 0.186,Y -583.644,Z 1479.220,A 0.000,B 0.000,C 90.000,E1 75.589} C_DIS
LIN {X -0.189,Y -584.519,Z 1479.213,A 0.000,B 0.000,C 90.000,E1 74.283} C_DIS
LIN {X -0.155,Y -585.446,Z 1479.204,A 0.000,B 0.000,C 90.000,E1 72.670} C_DIS
LIN {X -0.067,Y -586.524,Z 1479.193,A 0.000,B 0.000,C 90.000,E1 70.786} C_DIS
LIN {X 0.055,Y -587.461,Z 1479.183,A 0.000,B 0.000,C 90.000,E1 68.901} C_DIS
LIN {X -0.262,Y -588.717,Z 1479.171,A 0.000,B 0.000,C 90.000,E1 66.794} C_DIS
LIN {X 0.259,Y -589.560,Z 1479.164,A 0.000,B 0.000,C 90.000,E1 65.409} C_DIS
LIN {X -0.050,Y -590.756,Z 1479.152,A 0.000,B 0.000,C 90.000,E1 63.307} C_DIS
LIN {X -0.036,Y -591.667,Z 1479.144,A 0.000,B 0.000,C 90.000,E1 61.975} C_DIS
LIN {X -0.070,Y -592.934,Z 1479.135,A 0.000,B 0.000,C 90.000,E1 60.383} C_DIS
LIN {X 0.040,Y -594.641,Z 1479.124,A 0.000,B 0.000,C 90.000,E1 58.250} C_DIS
LIN {X 0.164,Y -595.725,Z 1479.116,A 0.000,B 0.000,C 90.000,E1 56.914} C_DIS
LIN {X 0.017,Y -597.075,Z 1479.108,A 0.000,B 0.000,C 90.000,E1 55.341} C_DIS
LIN {X -0.257,Y -598.256,Z 1479.099,A 0.000,B 0.000,C 90.000,E1 53.783} C_DIS
LIN {X 0.090,Y -599.187,Z 1479.091,A 0.000,B 0.000,C 90.000,E1 52.431} C_DIS
LIN {X 0.351,Y -599.855,Z 1479.084,A 0.000,B 0.000,C 90.000,E1 51.090} C_DIS
LIN {X -0.213,Y -600.500,Z 1479.077,A 0.000,B 0.000,C 90.000,E1 49.828} C_DIS
LIN {X 0.051,Y -600.835,Z 1479.072,A 0.000,B 0.000,C 90.000,E1 49.013} C_DIS
LIN {X -0.137,Y -600.995,Z 1479.068,A 0.000,B 0.000,C 90.000,E1 48.243} C_DIS
LIN {X 0.108,Y -601.059,Z 1479.061,A 0.000,B 0.000,C 90.000,E1 46.905} C_DIS
LIN {X -0.078,Y -601.019,Z 1479.056,A 0.000,B 0.000,C 90.000,E1 46.134} C_DIS
LIN {X -0.264,Y -600.763,Z 1479.049,A 0.000,B 0.000,C 90.000,E1 44.838} C_DIS
LIN {X -0.247,Y -600.272,Z 1479.043,A 0.000,B 0.000,C 90.000,E1 43.785} C_DIS
LIN {X -0.019,Y -599.355,Z 1479.036,A 0.000,B 0.000,C 90.000,E1 42.447} C_DIS
LIN {X -0.222,Y -598.668,Z 1479.031,A 0.000,B 0.000,C 90.000,E1 41.676} C_DIS
LIN {X -0.202,Y -597.524,Z 1479.026,A 0.000,B 0.000,C 90.000,E1 40.620} C_DIS
LIN {X -0.199,Y -596.162,Z 1479.020,A 0.000,B 0.000,C 90.000,E1 39.564} C_DIS
LIN {X 0.001,Y -594.246,Z 1479.012,A 0.000,B 0.000,C 90.000,E1 38.222} C_DIS
LIN {X 0.266,Y -591.951,Z 1479.005,A 0.000,B 0.000,C 90.000,E1 36.870} C_DIS
LIN {X 0.286,Y -589.750,Z 1478.999,A 0.000,B 0.000,C 90.000,E1 35.804} C_DIS
LIN {X 0.075,Y -587.883,Z 1478.995,A 0.000,B 0.000,C 90.000,E1 35.025} C_DIS
LIN {X -0.157,Y -585.776,Z 1478.990,A 0.000,B 0.000,C 90.000,E1 34.246} C_DIS
LIN {X 0.069,Y -583.363,Z 1478.986,A 0.000,B 0.000,C 90.000,E1 33.420} C_DIS
LIN {X 0.120,Y -579.782,Z 1478.980,A 0.000,B 0.000,C 90.000,E1 32.339} C_DIS
LIN {X 0.129,Y -577.744,Z 1478.977,A 0.000,B 0.000,C 90.000,E1 31.799} C_DIS
LIN {X -0.034,Y -574.284,Z 1478.972,A 0.000,B 0.000,C 90.000,E1 31.003} C_DIS
LIN {X -0.229,Y -570.491,Z 1478.968,A 0.000,B 0.000,C 90.000,E1 30.207} C_DIS
LIN {X 0.115,Y -566.989,Z 1478.964,A 0.000,B 0.000,C 90.000,E1 29.489} C_DIS
LIN {X -0.066,Y -563.354,Z 1478.960,A 0.000,B 0.000,C 90.000,E1 28.821} C_DIS
LIN {X 0.210,Y -559.413,Z 1478.956,A 0.000,B 0.000,C 90.000,E1 28.103} C_DIS
LIN {X -0.198,Y -555.937,Z 1478.953,A 0.000,B 0.000,C 90.000,E1 27.590} C_DIS
LIN {X -0.104,Y -550.330,Z 1478.949,A 0.000,B 0.000,C 90.000,E1 26.744} C_DIS
LIN {X 0.044,Y -547.280,Z 1478.946,A 0.000,B 0.000,C 90.000,E1 26.309} C_DIS
LIN {X -0.078,Y -543.842,Z 1478.944,A 0.000,B 0.000,C 90.000,E1 25.899} C_DIS
LIN {X 0.161,Y -541.222,Z 1478.942,A 0.000,B 0.000,C 90.000,E1 25.591} C_DIS
LIN {X 0.010,Y -538.214,Z 1478.941,A 0.000,B 0.000,C 90.000,E1 25.335} C_DIS
LIN {X -0.014,Y -536.518,Z 1478.940,A 0.000,B 0.000,C 90.000,E1 25.207} C_DIS
LIN {X 0.107,Y -534.772,Z 1478.939,A 0.000,B 0.000,C 90.000,E1 25.079} C_DIS
LIN {X 0.032,Y -531.702,Z 1478.939,A 0.000,B 0.000,C 90.000,E1 24.951} C_DIS
LIN {X -0.175,Y -530.556,Z 1478.939,A 0.000,B 0.000,C 90.000,E1 24.951} C_DIS
LIN {X 0.195,Y -382.994,Z 1478.939,A 0.000,B 0.000,C 90.000,E1 24.899} C_DIS
LIN {X 0.030,Y -378.917,Z 1478.924,A 0.000,B 0.000,C 90.000,E1 22.280} C_DIS
LIN {X 0.116,Y -373.676,Z 1478.898,A 0.000,B 0.000,C 90.000,E1 17.528} C_DIS
LIN {X -0.104,Y -368.073,Z 1478.869,A 0.000,B 0.000,C 90.000,E1 12.411} C_DIS
LIN {X 0.065,Y -366.388,Z 1478.854,A 0.000,B 0.000,C 90.000,E1 9.792} C_DIS
LIN {X 0.004,Y -361.734,Z 1478.821,A 0.000,B 0.000,C 90.000,E1 3.841} C_DIS
LIN {X -0.111,Y -360.854,Z 1478.801,A 0.000,B 0.000,C 90.000,E1 0.115} C_DIS
LIN {X -0.053,Y -359.426,Z 1478.770,A 0.000,B 0.000,C 90.000,E1 354.546} C_DIS
LIN {X 0.070,Y -358.890,Z 1478.759,A 0.000,B 0.000,C 90.000,E1 352.648} C_DIS
LIN {X -0.020,Y -359.563,Z 1478.726,A 0.000,B 0.000,C 90.000,E1 346.645} C_DIS
LIN {X 0.001,Y -361.801,Z 1478.684,A 0.000,B 0.000,C 90.000,E1 339.135} C_DIS
LIN {X -0.154,Y -362.053,Z 1478.680,A 0.000,B 0.000,C 90.000,E1 338.411} C_DIS
LIN {X 0.189,Y -365.980,Z 1478.643,A 0.000,B 0.000,C 90.000,E1 331.641} C_DIS
LIN {X 0.029,Y -366.387,Z 1478.639,A 0.000,B 0.000,C 90.000,E1 330.923} C_DIS
LIN {X -0.031,Y -371.355,Z 1478.604,A 0.000,B 0.000,C 90.000,E1 324.642} C_DIS
LIN {X -0.043,Y -371.766,Z 1478.602,A 0.000,B 0.000,C 90.000,E1 324.276} C_DIS
LIN {X 0.013,Y -377.358,Z 1478.567,A 0.000,B 0.000,C 90.000,E1 318.038} C_DIS
LIN {X 0.012,Y -378.235,Z 1478.563,A 0.000,B 0.000,C 90.000,E1 317.310} C_DIS
LIN {X 0.002,Y -383.940,Z 1478.531,A 0.000,B 0.000,C 90.000,E1 311.515} C_DIS
LIN {X 0.088,Y -384.893,Z 1478.527,A 0.000,B 0.000,C 90.000,E1 310.782} C_DIS
LIN {X 0.262,Y -390.610,Z 1478.495,A 0.000,B 0.000,C 90.000,E1 305.025} C_DIS
LIN {X 0.106,Y -391.104,Z 1478.493,A 0.000,B 0.000,C 90.000,E1 304.692} C_DIS
LIN {X 0.022,Y -391.648,Z 1478.489,A 0.000,B 0.000,C 90.000,E1 303.992} C_DIS
LIN {X -0.080,Y -396.825,Z 1478.459,A 0.000,B 0.000,C 90.000,E1 298.693} C_DIS
LIN {X -0.210,Y -397.120,Z 1478.457,A 0.000,B 0.000,C 90.000,E1 298.359} C_DIS
LIN {X -0.055,Y -401.597,Z 1478.426,A 0.000,B 0.000,C 90.000,E1 292.717} C_DIS
LIN {X 0.222,Y -404.659,Z 1478.395,A 0.000,B 0.000,C 90.000,E1 287.094} C_DIS
LIN {X -0.079,Y -404.735,Z 1478.391,A 0.000,B 0.000,C 90.000,E1 286.441} C_DIS
LIN {X 0.214,Y -406.099,Z 1478.364,A 0.000,B 0.000,C 90.000,E1 281.535} C_DIS
LIN {X -0.176,Y -406.094,Z 1478.362,A 0.000,B 0.000,C 90.000,E1 281.243} C_DIS
LIN {X -0.097,Y -405.680,Z 1478.333,A 0.000,B 0.000,C 90.000,E1 276.024} C_DIS
LIN {X -0.165,Y -405.058,Z 1478.328,A 0.000,B 0.000,C 90.000,E1 274.992} C_DIS
LIN {X -0.060,Y -403.497,Z 1478.304,A 0.000,B 0.000,C 90.000,E1 270.802} C_DIS
LIN {X -0.092,Y -403.288,Z 1478.302,A 0.000,B 0.000,C 90.000,E1 270.458} C_DIS
LIN {X 0.091,Y -398.931,Z 1478.271,A 0.000,B 0.000,C 90.000,E1 264.837} C_DIS
LIN {X -0.040,Y -393.108,Z 1478.242,A 0.000,B 0.000,C 90.000,E1 259.567} C_DIS
LIN {X -0.079,Y -392.835,Z 1478.240,A 0.000,B 0.000,C 90.000,E1 259.218} C_DIS
LIN {X 0.034,Y -385.993,Z 1478.212,A 0.000,B 0.000,C 90.000,E1 254.212} C_DIS
LIN {X -0.026,Y -385.267,Z 1478.208,A 0.000,B 0.000,C 90.000,E1 253.504} C_DIS
LIN {X -0.004,Y -384.768,Z 1478.206,A 0.000,B 0.000,C 90.000,E1 253.142} C_DIS
LIN {X 0.221,Y -377.973,Z 1478.182,A 0.000,B 0.000,C 90.000,E1 248.773} C_DIS
LIN {X -0.044,Y -376.233,Z 1478.174,A 0.000,B 0.000,C 90.000,E1 247.358} C_DIS
LIN {X 0.057,Y -374.944,Z 1478.170,A 0.000,B 0.000,C 90.000,E1 246.613} C_DIS
LIN {X -0.208,Y -368.417,Z 1478.148,A 0.000,B 0.000,C 90.000,E1 242.615} C_DIS
LIN {X 0.097,Y -366.047,Z 1478.137,A 0.000,B 0.000,C 90.000,E1 240.717} C_DIS
LIN {X 0.004,Y -359.196,Z 1478.115,A 0.000,B 0.000,C 90.000,E1 236.628} C_DIS
LIN {X 0.021,Y -355.842,Z 1478.100,A 0.000,B 0.000,C 90.000,E1 233.989} C_DIS
LIN {X -0.173,Y -348.793,Z 1478.075,A 0.000,B 0.000,C 90.000,E1 229.461} C_DIS
LIN {X -0.097,Y -346.185,Z 1478.062,A 0.000,B 0.000,C 90.000,E1 227.148} C_DIS
LIN {X -0.088,Y -345.065,Z 1478.058,A 0.000,B 0.000,C 90.000,E1 226.377} C_DIS
LIN {X 0.094,Y -338.586,Z 1478.030,A 0.000,B 0.000,C 90.000,E1 221.310} C_DIS
LIN {X 0.094,Y -336.840,Z 1478.019,A 0.000,B 0.000,C 90.000,E1 219.358} C_DIS
LIN {X 0.014,Y -330.861,Z 1477.988,A 0.000,B 0.000,C 90.000,E1 213.865} C_DIS
LIN {X 0.149,Y -329.296,Z 1477.975,A 0.000,B 0.000,C 90.000,E1 211.465} C_DIS
LIN {X -0.154,Y -324.669,Z 1477.942,A 0.000,B 0.000,C 90.000,E1 205.540} C_DIS
LIN {X 0.174,Y -323.837,Z 1477.928,A 0.000,B 0.000,C 90.000,E1 203.078} C_DIS
LIN {X -0.017,Y -321.124,Z 1477.881,A 0.000,B 0.000,C 90.000,E1 194.662} C_DIS
LIN {X 0.138,Y -320.932,Z 1477.877,A 0.000,B 0.000,C 90.000,E1 193.828} C_DIS
LIN {X -0.076,Y -321.562,Z 1477.832,A 0.000,B 0.000,C 90.000,E1 185.796} C_DIS
LIN {X -0.143,Y -324.415,Z 1477.790,A 0.000,B 0.000,C 90.000,E1 178.165} C_DIS
LIN {X -0.141,Y -325.376,Z 1477.783,A 0.000,B 0.000,C 90.000,E1 176.963} C_DIS
LIN {X -0.100,Y -329.112,Z 1477.750,A 0.000,B 0.000,C 90.000,E1 170.971} C_DIS
LIN {X 0.061,Y -334.260,Z 1477.726,A 0.000,B 0.000,C 90.000,E1 166.589} C_DIS
LIN {X 0.067,Y -335.488,Z 1477.719,A 0.000,B 0.000,C 90.000,E1 165.408} C_DIS
LIN {X 0.143,Y -340.932,Z 1477.695,A 0.000,B 0.000,C 90.000,E1 161.094} C_DIS
LIN {X -0.172,Y -342.138,Z 1477.691,A 0.000,B 0.000,C 90.000,E1 160.369} C_DIS
LIN {X -0.058,Y -347.939,Z 1477.667,A 0.000,B 0.000,C 90.000,E1 156.102} C_DIS
LIN {X -0.055,Y -352.455,Z 1477.653,A 0.000,B 0.000,C 90.000,E1 153.563} C_DIS
LIN {X -0.123,Y -492.548,Z 1477.653,A 0.000,B 0.000,C 90.000,E1 153.563} C_DIS
LIN {X 0.155,Y -495.416,Z 1477.653,A 0.000,B 0.000,C 90.000,E1 153.461} C_DIS
LIN {X 0.261,Y -496.880,Z 1477.652,A 0.000,B 0.000,C 90.000,E1 153.384} C_DIS
LIN {X 0.049,Y -499.607,Z 1477.651,A 0.000,B 0.000,C 90.000,E1 153.256} C_DIS
LIN {X -0.005,Y -502.191,Z 1477.651,A 0.000,B 0.000,C 90.000,E1 153.076} C_DIS
LIN {X -0.151,Y -506.187,Z 1477.649,A 0.000,B 0.000,C 90.000,E1 152.743} C_DIS
LIN {X -0.323,Y -509.945,Z 1477.646,A 0.000,B 0.000,C 90.000,E1 152.359} C_DIS
LIN {X 0.019,Y -512.377,Z 1477.645,A 0.000,B 0.000,C 90.000,E1 152.025} C_DIS
LIN {X 0.011,Y -516.564,Z 1477.641,A 0.000,B 0.000,C 90.000,E1 151.435} C_DIS
LIN {X 0.037,Y -520.271,Z 1477.638,A 0.000,B 0.000,C 90.000,E1 150.845} C_DIS
LIN {X 0.088,Y -523.560,Z 1477.635,A 0.000,B 0.000,C 90.000,E1 150.255} C_DIS
LIN {X 0.007,Y -527.247,Z 1477.631,A 0.000,B 0.000,C 90.000,E1 149.537} C_DIS
LIN {X 0.226,Y -530.455,Z 1477.627,A 0.000,B 0.000,C 90.000,E1 148.791} C_DIS
LIN {X -0.103,Y -532.828,Z 1477.624,A 0.000,B 0.000,C 90.000,E1 148.250} C_DIS
LIN {X 0.031,Y -534.917,Z 1477.620,A 0.000,B 0.000,C 90.000,E1 147.661} C_DIS
LIN {X -0.278,Y -537.758,Z 1477.616,A 0.000,B 0.000,C 90.000,E1 146.834} C_DIS
LIN {X -0.109,Y -540.344,Z 1477.611,A 0.000,B 0.000,C 90.000,E1 145.960} C_DIS
LIN {X -0.055,Y -542.759,Z 1477.606,A 0.000,B 0.000,C 90.000,E1 145.102} C_DIS
LIN {X -0.284,Y -544.906,Z 1477.601,A 0.000,B 0.000,C 90.000,E1 144.276} C_DIS
LIN {X -0.174,Y -546.755,Z 1477.597,A 0.000,B 0.000,C 90.000,E1 143.417} C_DIS
LIN {X 0.006,Y -548.929,Z 1477.590,A 0.000,B 0.000,C 90.000,E1 142.271} C_DIS
LIN {X -0.271,Y -550.373,Z 1477.586,A 0.000,B 0.000,C 90.000,E1 141.457} C_DIS
LIN {X 0.303,Y -552.008,Z 1477.580,A 0.000,B 0.000,C 90.000,E1 140.275} C_DIS
LIN {X 0.119,Y -553.536,Z 1477.573,A 0.000,B 0.000,C 90.000,E1 139.175} C_DIS
LIN {X -0.103,Y -554.831,Z 1477.567,A 0.000,B 0.000,C 90.000,E1 138.081} C_DIS
LIN {X 0.142,Y -556.310,Z 1477.559,A 0.000,B 0.000,C 90.000,E1 136.662} C_DIS
LIN {X 0.021,Y -557.590,Z 1477.552,A 0.000,B 0.000,C 90.000,E1 135.283} C_DIS
LIN {X -0.033,Y -558.869,Z 1477.542,A 0.000,B 0.000,C 90.000,E1 133.623} C_DIS
LIN {X -0.177,Y -559.569,Z 1477.536,A 0.000,B 0.000,C 90.000,E1 132.528} C_DIS
LIN {X 0.021,Y -559.981,Z 1477.532,A 0.000,B 0.000,C 90.000,E1 131.676} C_DIS
LIN {X 0.309,Y -560.349,Z 1477.525,A 0.000,B 0.000,C 90.000,E1 130.539} C_DIS
LIN {X -0.097,Y -560.608,Z 1477.518,A 0.000,B 0.000,C 90.000,E1 129.197} C_DIS
LIN {X -0.159,Y -560.771,Z 1477.512,A 0.000,B 0.000,C 90.000,E1 128.096} C_DIS
LIN {X -0.127,Y -560.917,Z 1477.504,A 0.000,B 0.000,C 90.000,E1 126.710} C_DIS
LIN {X -0.074,Y -560.943,Z 1477.498,A 0.000,B 0.000,C 90.000,E1 125.598} C_DIS
LIN {X -0.013,Y -560.755,Z 1477.492,A 0.000,B 0.000,C 90.000,E1 124.485} C_DIS
LIN {X -0.039,Y -560.454,Z 1477.476,A 0.000,B 0.000,C 90.000,E1 121.720} C_DIS
LIN {X -0.156,Y -560.563,Z 1477.465,A 0.000,B 0.000,C 90.000,E1 119.795} C_DIS
LIN {X -0.050,Y -560.846,Z 1477.455,A 0.000,B 0.000,C 90.000,E1 117.847} C_DIS
LIN {X 0.060,Y -561.213,Z 1477.444,A 0.000,B 0.000,C 90.000,E1 115.899} C_DIS
LIN {X -0.125,Y -561.593,Z 1477.435,A 0.000,B 0.000,C 90.000,E1 114.259} C_DIS
LIN {X 0.097,Y -562.015,Z 1477.429,A 0.000,B 0.000,C 90.000,E1 113.131} C_DIS
LIN {X -0.189,Y -562.572,Z 1477.418,A 0.000,B 0.000,C 90.000,E1 111.227} C_DIS
LIN {X 0.072,Y -563.050,Z 1477.407,A 0.000,B 0.000,C 90.000,E1 109.268} C_DIS
LIN {X 0.227,Y -563.400,Z 1477.400,A 0.000,B 0.000,C 90.000,E1 107.873} C_DIS
LIN {X -0.022,Y -563.939,Z 1477.389,A 0.000,B 0.000,C 90.000,E1 105.969} C_DIS
LIN {X -0.252,Y -564.571,Z 1477.378,A 0.000,B 0.000,C 90.000,E1 104.064} C_DIS
LIN {X 0.099,Y -565.430,Z 1477.366,A 0.000,B 0.000,C 90.000,E1 101.827} C_DIS
LIN {X -0.271,Y -565.964,Z 1477.358,A 0.000,B 0.000,C 90.000,E1 100.489} C_DIS
LIN {X 0.276,Y -566.847,Z 1477.348,A 0.000,B 0.000,C 90.000,E1 98.511} C_DIS
LIN {X 0.286,Y -567.934,Z 1477.335,A 0.000,B 0.000,C 90.000,E1 96.315} C_DIS
LIN {X 0.095,Y -569.100,Z 1477.325,A 0.000,B 0.000,C 90.000,E1 94.416} C_DIS
LIN {X -0.110,Y -570.390,Z 1477.314,A 0.000,B 0.000,C 90.000,E1 92.522} C_DIS
LIN {X -0.007,Y -571.379,Z 1477.306,A 0.000,B 0.000,C 90.000,E1 91.146} C_DIS
LIN {X 0.240,Y -572.577,Z 1477.297,A 0.000,B 0.000,C 90.000,E1 89.484} C_DIS
LIN {X -0.189,Y -573.625,Z 1477.290,A 0.000,B 0.000,C 90.000,E1 88.165} C_DIS
LIN {X 0.122,Y -574.864,Z 1477.281,A 0.000,B 0.000,C 90.000,E1 86.502} C_DIS
LIN {X 0.053,Y -576.315,Z 1477.270,A 0.000,B 0.000,C 90.000,E1 84.609} C_DIS
LIN {X -0.084,Y -577.613,Z 1477.261,A 0.000,B 0.000,C 90.000,E1 82.996} C_DIS
LIN {X -0.251,Y -578.753,Z 1477.254,A 0.000,B 0.000,C 90.000,E1 81.659} C_DIS
LIN {X 0.093,Y -579.885,Z 1477.246,A 0.000,B 0.000,C 90.000,E1 80.274} C_DIS
LIN {X 0.080,Y -581.037,Z 1477.239,A 0.000,B 0.000,C 90.000,E1 78.926} C_DIS
LIN {X -0.129,Y -582.720,Z 1477.228,A 0.000,B 0.000,C 90.000,E1 77.061} C_DIS
LIN {X 0.045,Y -583.786,Z 1477.221,A 0.000,B 0.000,C 90.000,E1 75.700} C_DIS
LIN {X 0.240,Y -584.667,Z 1477.213,A 0.000,B 0.000,C 90.000,E1 74.338} C_DIS
LIN {X 0.282,Y -585.578,Z 1477.204,A 0.000,B 0.000,C 90.000,E1 72.725} C_DIS
LIN {X 0.050,Y -586.810,Z 1477.192,A 0.000,B 0.000,C 90.000,E1 70.604} C_DIS
LIN {X 0.176,Y -587.763,Z 1477.182,A 0.000,B 0.000,C 90.000,E1 68.720} C_DIS
LIN {X -0.137,Y -589.013,Z 1477.170,A 0.000,B 0.000,C 90.000,E1 66.613} C_DIS
LIN {X -0.150,Y -589.848,Z 1477.163,A 0.000,B 0.000,C 90.000,E1 65.281} C_DIS
LIN {X 0.078,Y -591.085,Z 1477.151,A 0.000,B 0.000,C 90.000,E1 63.127} C_DIS
LIN {X 0.065,Y -592.645,Z 1477.139,A 0.000,B 0.000,C 90.000,E1 61.001} C_DIS
LIN {X 0.050,Y -593.913,Z 1477.130,A 0.000,B 0.000,C 90.000,E1 59.410} C_DIS
LIN {X 0.373,Y -595.236,Z 1477.121,A 0.000,B 0.000,C 90.000,E1 57.788} C_DIS
LIN {X 0.001,Y -596.331,Z 1477.114,A 0.000,B 0.000,C 90.000,E1 56.501} C_DIS
LIN {X 0.207,Y -597.638,Z 1477.105,A 0.000,B 0.000,C 90.000,E1 54.895} C_DIS
LIN {X -0.284,Y -598.598,Z 1477.098,A 0.000,B 0.000,C 90.000,E1 53.623} C_DIS
LIN {X 0.076,Y -599.493,Z 1477.090,A 0.000,B 0.000,C 90.000,E1 52.271} C_DIS
LIN {X -0.031,Y -600.232,Z 1477.083,A 0.000,B 0.000,C 90.000,E1 50.964} C_DIS
LIN {X 0.011,Y -600.734,Z 1477.077,A 0.000,B 0.000,C 90.000,E1 49.908} C_DIS
LIN {X -0.178,Y -601.074,Z 1477.073,A 0.000,B 0.000,C 90.000,E1 49.138} C_DIS
LIN {X -0.122,Y -601.250,Z 1477.067,A 0.000,B 0.000,C 90.000,E1 48.081} C_DIS
LIN {X -0.073,Y -601.343,Z 1477.061,A 0.000,B 0.000,C 90.000,E1 47.025} C_DIS
LIN {X 0.154,Y -601.329,Z 1477.057,A 0.000,B 0.000,C 90.000,E1 46.215} C_DIS
LIN {X 0.179,Y -601.171,Z 1477.051,A 0.000,B 0.000,C 90.000,E1 45.162} C_DIS
LIN {X -0.005,Y -600.633,Z 1477.044,A 0.000,B 0.000,C 90.000,E1 43.866} C_DIS
LIN {X 0.230,Y -599.744,Z 1477.036,A 0.000,B 0.000,C 90.000,E1 42.528} C_DIS
LIN {X -0.186,Y -598.787,Z 1477.031,A 0.000,B 0.000,C 90.000,E1 41.515} C_DIS
LIN {X 0.057,Y -597.948,Z 1477.026,A 0.000,B 0.000,C 90.000,E1 40.701} C_DIS
LIN {X 0.068,Y -596.623,Z 1477.020,A 0.000,B 0.000,C 90.000,E1 39.644} C_DIS
LIN {X -0.092,Y -594.711,Z 1477.013,A 0.000,B 0.000,C 90.000,E1 38.338} C_DIS
LIN {X 0.077,Y -592.457,Z 1477.006,A 0.000,B 0.000,C 90.000,E1 36.996} C_DIS
LIN {X 0.101,Y -590.342,Z 1477.000,A 0.000,B 0.000,C 90.000,E1 35.931} C_DIS
LIN {X -0.105,Y -588.511,Z 1476.995,A 0.000,B 0.000,C 90.000,E1 35.152} C_DIS
LIN {X -0.044,Y -587.166,Z 1476.992,A 0.000,B 0.000,C 90.000,E1 34.612} C_DIS
LIN {X 0.202,Y -584.896,Z 1476.988,A 0.000,B 0.000,C 90.000,E1 33.785} C_DIS
LIN {X -0.242,Y -583.247,Z 1476.985,A 0.000,B 0.000,C 90.000,E1 33.293} C_DIS
LIN {X -0.187,Y -579.626,Z 1476.979,A 0.000,B 0.000,C 90.000,E1 32.212} C_DIS
LIN {X -0.178,Y -577.570,Z 1476.976,A 0.000,B 0.000,C 90.000,E1 31.671} C_DIS
LIN {X -0.045,Y -574.078,Z 1476.971,A 0.000,B 0.000,C 90.000,E1 30.846} C_DIS
LIN {X 0.245,Y -570.261,Z 1476.967,A 0.000,B 0.000,C 90.000,E1 30.001} C_DIS
LIN {X -0.277,Y -563.800,Z 1476.960,A 0.000,B 0.000,C 90.000,E1 28.821} C_DIS
LIN {X -0.094,Y -559.048,Z 1476.955,A 0.000,B 0.000,C 90.000,E1 27.975} C_DIS
LIN {X 0.142,Y -554.621,Z 1476.952,A 0.000,B 0.000,C 90.000,E1 27.257} C_DIS
LIN {X 0.083,Y -549.904,Z 1476.948,A 0.000,B 0.000,C 90.000,E1 26.565} C_DIS
LIN {X 0.105,Y -543.788,Z 1476.943,A 0.000,B 0.000,C 90.000,E1 25.720} C_DIS
LIN {X 0.217,Y -540.202,Z 1476.941,A 0.000,B 0.000,C 90.000,E1 25.283} C_DIS
LIN {X -0.033,Y -537.447,Z 1476.939,A 0.000,B 0.000,C 90.000,E1 25.027} C_DIS
LIN {X -0.146,Y -534.371,Z 1476.938,A 0.000,B 0.000,C 90.000,E1 24.771} C_DIS
LIN {X -0.086,Y -532.773,Z 1476.937,A 0.000,B 0.000,C 90.000,E1 24.643} C_DIS
LIN {X -0.001,Y -529.925,Z 1476.936,A 0.000,B 0.000,C 90.000,E1 24.463} C_DIS
LIN {X -0.051,Y -527.871,Z 1476.936,A 0.000,B 0.000,C 90.000,E1 24.387} C_DIS
LIN {X 0.199,Y -526.598,Z 1476.935,A 0.000,B 0.000,C 90.000,E1 24.335} C_DIS
LIN {X 0.121,Y -382.097,Z 1476.935,A 0.000,B 0.000,C 90.000,E1 24.335} C_DIS
LIN {X 0.104,Y -375.599,Z 1476.909,A 0.000,B 0.000,C 90.000,E1 19.577} C_DIS
LIN {X -0.017,Y -373.522,Z 1476.897,A 0.000,B 0.000,C 90.000,E1 17.402} C_DIS
LIN {X 0.022,Y -367.957,Z 1476.868,A 0.000,B 0.000,C 90.000,E1 12.243} C_DIS
LIN {X 0.041,Y -366.538,Z 1476.856,A 0.000,B 0.000,C 90.000,E1 10.018} C_DIS
LIN {X -0.031,Y -365.426,Z 1476.850,A 0.000,B 0.000,C 90.000,E1 8.916} C_DIS
LIN {X -0.066,Y -361.273,Z 1476.814,A 0.000,B 0.000,C 90.000,E1 2.579} C_DIS
LIN {X -0.140,Y -360.906,Z 1476.802,A 0.000,B 0.000,C 90.000,E1 0.344} C_DIS
LIN {X -0.157,Y -359.667,Z 1476.784,A 0.000,B 0.000,C 90.000,E1 357.192} C_DIS
LIN {X -0.053,Y -359.426,Z 1476.770,A 0.000,B 0.000,C 90.000,E1 354.546} C_DIS
LIN {X 0.070,Y -358.890,Z 1476.759,A 0.000,B 0.000,C 90.000,E1 352.648} C_DIS
LIN {X -0.020,Y -359.563,Z 1476.726,A 0.000,B 0.000,C 90.000,E1 346.645} C_DIS
LIN {X 0.001,Y -361.801,Z 1476.684,A 0.000,B 0.000,C 90.000,E1 339.135} C_DIS
LIN {X -0.154,Y -362.053,Z 1476.680,A 0.000,B 0.000,C 90.000,E1 338.411} C_DIS
LIN {X 0.189,Y -365.980,Z 1476.643,A 0.000,B 0.000,C 90.000,E1 331.641} C_DIS
LIN {X 0.029,Y -366.387,Z 1476.639,A 0.000,B 0.000,C 90.000,E1 330.923} C_DIS
LIN {X -0.031,Y -371.355,Z 1476.604,A 0.000,B 0.000,C 90.000,E1 324.642} C_DIS
LIN {X -0.043,Y -371.766,Z 1476.602,A 0.000,B 0.000,C 90.000,E1 324.276} C_DIS
LIN {X 0.013,Y -377.358,Z 1476.567,A 0.000,B 0.000,C 90.000,E1 318.038} C_DIS
LIN {X 0.012,Y -378.235,Z 1476.563,A 0.000,B 0.000,C 90.000,E1 317.310} C_DIS
LIN {X 0.002,Y -383.940,Z 1476.531,A 0.000,B 0.000,C 90.000,E1 311.515} C_DIS
LIN {X 0.088,Y -384.893,Z 1476.527,A 0.000,B 0.000,C 90.000,E1 310.782} C_DIS
LIN {X 0.262,Y -390.610,Z 1476.495,A 0.000,B 0.000,C 90.000,E1 305.025} C_DIS
LIN {X 0.106,Y -391.104,Z 1476.493,A 0.000,B 0.000,C 90.000,E1 304.692} C_DIS
LIN {X 0.022,Y -391.648,Z 1476.489,A 0.000,B 0.000,C 90.000,E1 303.992} C_DIS
LIN {X -0.080,Y -396.825,Z 1476.459,A 0.000,B 0.000,C 90.000,E1 298.693} C_DIS
LIN {X -0.210,Y -397.120,Z 1476.457,A 0.000,B 0.000,C 90.000,E1 298.359} C_DIS
LIN {X -0.055,Y -401.597,Z 1476.426,A 0.000,B 0.000,C 90.000,E1 292.717} C_DIS
LIN {X 0.222,Y -404.659,Z 1476.395,A 0.000,B 0.000,C 90.000,E1 287.094} C_DIS
LIN {X -0.079,Y -404.735,Z 1476.391,A 0.000,B 0.000,C 90.000,E1 286.441} C_DIS
LIN {X 0.214,Y -406.099,Z 1476.364,A 0.000,B 0.000,C 90.000,E1 281.535} C_DIS
LIN {X -0.176,Y -406.094,Z 1476.362,A 0.000,B 0.000,C 90.000,E1 281.243} C_DIS
LIN {X -0.097,Y -405.680,Z 1476.333,A 0.000,B 0.000,C 90.000,E1 276.024} C_DIS
LIN {X -0.165,Y -405.058,Z 1476.328,A 0.000,B 0.000,C 90.000,E1 274.992} C_DIS
LIN {X -0.060,Y -403.497,Z 1476.304,A 0.000,B 0.000,C 90.000,E1 270.802} C_DIS
LIN {X -0.092,Y -403.288,Z 1476.302,A 0.000,B 0.000,C 90.000,E1 270.458} C_DIS
LIN {X 0.091,Y -398.931,Z 1476.271,A 0.000,B 0.000,C 90.000,E1 264.837} C_DIS
LIN {X -0.040,Y -393.108,Z 1476.242,A 0.000,B 0.000,C 90.000,E1 259.567} C_DIS
LIN {X -0.079,Y -392.835,Z 1476.240,A 0.000,B 0.000,C 90.000,E1 259.218} C_DIS
LIN {X 0.034,Y -385.993,Z 1476.212,A 0.000,B 0.000,C 90.000,E1 254.212} C_DIS
LIN {X -0.026,Y -385.267,Z 1476.208,A 0.000,B 0.000,C 90.000,E1 253.504} C_DIS
LIN {X -0.004,Y -384.768,Z 1476.206,A 0.000,B 0.000,C 90.000,E1 253.142} C_DIS
LIN {X 0.221,Y -377.973,Z 1476.182,A 0.000,B 0.000,C 90.000,E1 248.773} C_DIS
LIN {X -0.044,Y -376.233,Z 1476.174,A 0.000,B 0.000,C 90.000,E1 247.358} C_DIS
LIN {X 0.057,Y -374.944,Z 1476.170,A 0.000,B 0.000,C 90.000,E1 246.613} C_DIS
LIN {X -0.208,Y -368.417,Z 1476.148,A 0.000,B 0.000,C 90.000,E1 242.615} C_DIS
LIN {X 0.097,Y -366.047,Z 1476.137,A 0.000,B 0.000,C 90.000,E1 240.717} C_DIS
LIN {X 0.004,Y -359.196,Z 1476.115,A 0.000,B 0.000,C 90.000,E1 236.628} C_DIS
LIN {X 0.021,Y -355.842,Z 1476.100,A 0.000,B 0.000,C 90.000,E1 233.989} C_DIS
LIN {X -0.173,Y -348.793,Z 1476.075,A 0.000,B 0.000,C 90.000,E1 229.461} C_DIS
LIN {X -0.097,Y -346.185,Z 1476.062,A 0.000,B 0.000,C 90.000,E1 227.148} C_DIS
LIN {X -0.088,Y -345.065,Z 1476.058,A 0.000,B 0.000,C 90.000,E1 226.377} C_DIS
LIN {X 0.094,Y -338.586,Z 1476.030,A 0.000,B 0.000,C 90.000,E1 221.310} C_DIS
LIN {X 0.094,Y -336.840,Z 1476.019,A 0.000,B 0.000,C 90.000,E1 219.358} C_DIS
LIN {X 0.014,Y -330.861,Z 1475.988,A 0.000,B 0.000,C 90.000,E1 213.865} C_DIS
LIN {X 0.149,Y -329.296,Z 1475.975,A 0.000,B 0.000,C 90.000,E1 211.465} C_DIS
LIN {X -0.154,Y -324.669,Z 1475.942,A 0.000,B 0.000,C 90.000,E1 205.540} C_DIS
LIN {X 0.174,Y -323.837,Z 1475.928,A 0.000,B 0.000,C 90.000,E1 203.078} C_DIS
LIN {X -0.017,Y -321.124,Z 1475.881,A 0.000,B 0.000,C 90.000,E1 194.662} C_DIS
LIN {X 0.138,Y -320.932,Z 1475.877,A 0.000,B 0.000,C 90.000,E1 193.828} C_DIS
LIN {X -0.076,Y -321.562,Z 1475.832,A 0.000,B 0.000,C 90.000,E1 185.796} C_DIS
LIN {X -0.143,Y -324.415,Z 1475.790,A 0.000,B 0.000,C 90.000,E1 178.165} C_DIS
LIN {X -0.141,Y -325.376,Z 1475.783,A 0.000,B 0.000,C 90.000,E1 176.963} C_DIS
LIN {X -0.100,Y -329.112,Z 1475.750,A 0.000,B 0.000,C 90.000,E1 170.971} C_DIS
LIN {X 0.061,Y -334.260,Z 1475.726,A 0.000,B 0.000,C 90.000,E1 166.589} C_DIS
LIN {X 0.067,Y -335.488,Z 1475.719,A 0.000,B 0.000,C 90.000,E1 165.408} C_DIS
LIN {X 0.143,Y -340.932,Z 1475.695,A 0.000,B 0.000,C 90.000,E1 161.094} C_DIS
LIN {X -0.172,Y -342.138,Z 1475.691,A 0.000,B 0.000,C 90.000,E1 160.369} C_DIS
LIN {X -0.058,Y -347.939,Z 1475.667,A 0.000,B 0.000,C 90.000,E1 156.102} C_DIS
LIN {X 0.087,Y -351.386,Z 1475.656,A 0.000,B 0.000,C 90.000,E1 154.101} C_DIS
LIN {X 0.073,Y -487.346,Z 1475.656,A 0.000,B 0.000,C 90.000,E1 154.101} C_DIS
LIN {X 0.024,Y -488.055,Z 1475.656,A 0.000,B 0.000,C 90.000,E1 154.101} C_DIS
LIN {X 0.064,Y -490.746,Z 1475.656,A 0.000,B 0.000,C 90.000,E1 154.024} C_DIS
LIN {X 0.104,Y -492.410,Z 1475.655,A 0.000,B 0.000,C 90.000,E1 153.948} C_DIS
LIN {X 0.232,Y -495.392,Z 1475.654,A 0.000,B 0.000,C 90.000,E1 153.768} C_DIS
LIN {X -0.253,Y -498.101,Z 1475.653,A 0.000,B 0.000,C 90.000,E1 153.640} C_DIS
LIN {X 0.166,Y -502.232,Z 1475.652,A 0.000,B 0.000,C 90.000,E1 153.256} C_DIS
LIN {X 0.091,Y -506.099,Z 1475.649,A 0.000,B 0.000,C 90.000,E1 152.871} C_DIS
LIN {X 0.084,Y -509.784,Z 1475.647,A 0.000,B 0.000,C 90.000,E1 152.436} C_DIS
LIN {X -0.222,Y -513.217,Z 1475.645,A 0.000,B 0.000,C 90.000,E1 152.025} C_DIS
LIN {X 0.229,Y -517.328,Z 1475.641,A 0.000,B 0.000,C 90.000,E1 151.385} C_DIS
LIN {X 0.258,Y -520.986,Z 1475.638,A 0.000,B 0.000,C 90.000,E1 150.795} C_DIS
LIN {X -0.140,Y -524.247,Z 1475.635,A 0.000,B 0.000,C 90.000,E1 150.255} C_DIS
LIN {X -0.218,Y -527.858,Z 1475.631,A 0.000,B 0.000,C 90.000,E1 149.537} C_DIS
LIN {X -0.114,Y -530.509,Z 1475.627,A 0.000,B 0.000,C 90.000,E1 148.948} C_DIS
LIN {X 0.132,Y -533.407,Z 1475.623,A 0.000,B 0.000,C 90.000,E1 148.201} C_DIS
LIN {X -0.193,Y -536.400,Z 1475.619,A 0.000,B 0.000,C 90.000,E1 147.375} C_DIS
LIN {X -0.034,Y -539.187,Z 1475.614,A 0.000,B 0.000,C 90.000,E1 146.501} C_DIS
LIN {X -0.279,Y -542.442,Z 1475.608,A 0.000,B 0.000,C 90.000,E1 145.388} C_DIS
LIN {X 0.281,Y -545.335,Z 1475.601,A 0.000,B 0.000,C 90.000,E1 144.196} C_DIS
LIN {X 0.072,Y -547.171,Z 1475.597,A 0.000,B 0.000,C 90.000,E1 143.371} C_DIS
LIN {X -0.180,Y -549.337,Z 1475.590,A 0.000,B 0.000,C 90.000,E1 142.271} C_DIS
LIN {X 0.030,Y -551.150,Z 1475.584,A 0.000,B 0.000,C 90.000,E1 141.126} C_DIS
LIN {X 0.185,Y -552.740,Z 1475.578,A 0.000,B 0.000,C 90.000,E1 139.989} C_DIS
LIN {X 0.369,Y -554.161,Z 1475.572,A 0.000,B 0.000,C 90.000,E1 138.852} C_DIS
LIN {X 0.162,Y -555.413,Z 1475.565,A 0.000,B 0.000,C 90.000,E1 137.757} C_DIS
LIN {X -0.024,Y -556.548,Z 1475.559,A 0.000,B 0.000,C 90.000,E1 136.662} C_DIS
LIN {X -0.199,Y -557.542,Z 1475.553,A 0.000,B 0.000,C 90.000,E1 135.567} C_DIS
LIN {X 0.145,Y -558.858,Z 1475.544,A 0.000,B 0.000,C 90.000,E1 133.866} C_DIS
LIN {X -0.120,Y -559.205,Z 1475.541,A 0.000,B 0.000,C 90.000,E1 133.338} C_DIS
LIN {X -0.333,Y -559.713,Z 1475.536,A 0.000,B 0.000,C 90.000,E1 132.528} C_DIS
LIN {X -0.049,Y -560.202,Z 1475.530,A 0.000,B 0.000,C 90.000,E1 131.391} C_DIS
LIN {X -0.181,Y -560.531,Z 1475.524,A 0.000,B 0.000,C 90.000,E1 130.297} C_DIS
LIN {X -0.060,Y -560.782,Z 1475.515,A 0.000,B 0.000,C 90.000,E1 128.624} C_DIS
LIN {X 0.173,Y -560.982,Z 1475.504,A 0.000,B 0.000,C 90.000,E1 126.664} C_DIS
LIN {X -0.222,Y -561.008,Z 1475.498,A 0.000,B 0.000,C 90.000,E1 125.598} C_DIS
LIN {X -0.066,Y -560.696,Z 1475.490,A 0.000,B 0.000,C 90.000,E1 124.199} C_DIS
LIN {X 0.291,Y -560.455,Z 1475.476,A 0.000,B 0.000,C 90.000,E1 121.671} C_DIS
LIN {X 0.183,Y -560.539,Z 1475.465,A 0.000,B 0.000,C 90.000,E1 119.745} C_DIS
LIN {X 0.003,Y -560.809,Z 1475.456,A 0.000,B 0.000,C 90.000,E1 118.103} C_DIS
LIN {X 0.063,Y -561.087,Z 1475.447,A 0.000,B 0.000,C 90.000,E1 116.437} C_DIS
LIN {X -0.072,Y -561.562,Z 1475.436,A 0.000,B 0.000,C 90.000,E1 114.515} C_DIS
LIN {X 0.266,Y -562.094,Z 1475.427,A 0.000,B 0.000,C 90.000,E1 112.823} C_DIS
LIN {X -0.335,Y -562.607,Z 1475.418,A 0.000,B 0.000,C 90.000,E1 111.227} C_DIS
LIN {X 0.243,Y -563.159,Z 1475.406,A 0.000,B 0.000,C 90.000,E1 108.960} C_DIS
LIN {X 0.226,Y -563.490,Z 1475.398,A 0.000,B 0.000,C 90.000,E1 107.583} C_DIS
LIN {X -0.167,Y -563.975,Z 1475.389,A 0.000,B 0.000,C 90.000,E1 105.969} C_DIS
LIN {X 0.152,Y -564.607,Z 1475.378,A 0.000,B 0.000,C 90.000,E1 104.008} C_DIS
LIN {X -0.044,Y -565.468,Z 1475.366,A 0.000,B 0.000,C 90.000,E1 101.827} C_DIS
LIN {X -0.243,Y -566.124,Z 1475.357,A 0.000,B 0.000,C 90.000,E1 100.197} C_DIS
LIN {X 0.134,Y -566.886,Z 1475.347,A 0.000,B 0.000,C 90.000,E1 98.511} C_DIS
LIN {X 0.146,Y -567.976,Z 1475.335,A 0.000,B 0.000,C 90.000,E1 96.315} C_DIS
LIN {X -0.161,Y -568.950,Z 1475.326,A 0.000,B 0.000,C 90.000,E1 94.702} C_DIS
LIN {X -0.212,Y -569.666,Z 1475.320,A 0.000,B 0.000,C 90.000,E1 93.612} C_DIS
LIN {X 0.013,Y -570.889,Z 1475.311,A 0.000,B 0.000,C 90.000,E1 91.949} C_DIS
LIN {X -0.035,Y -572.486,Z 1475.299,A 0.000,B 0.000,C 90.000,E1 89.771} C_DIS
LIN {X 0.091,Y -573.542,Z 1475.291,A 0.000,B 0.000,C 90.000,E1 88.396} C_DIS
LIN {X -0.010,Y -574.988,Z 1475.281,A 0.000,B 0.000,C 90.000,E1 86.502} C_DIS
LIN {X -0.077,Y -576.455,Z 1475.270,A 0.000,B 0.000,C 90.000,E1 84.609} C_DIS
LIN {X -0.002,Y -578.011,Z 1475.260,A 0.000,B 0.000,C 90.000,E1 82.704} C_DIS
LIN {X 0.199,Y -578.924,Z 1475.254,A 0.000,B 0.000,C 90.000,E1 81.602} C_DIS
LIN {X -0.029,Y -580.081,Z 1475.246,A 0.000,B 0.000,C 90.000,E1 80.274} C_DIS
LIN {X -0.039,Y -581.217,Z 1475.239,A 0.000,B 0.000,C 90.000,E1 78.926} C_DIS
LIN {X -0.243,Y -582.923,Z 1475.228,A 0.000,B 0.000,C 90.000,E1 77.061} C_DIS
LIN {X -0.066,Y -584.013,Z 1475.221,A 0.000,B 0.000,C 90.000,E1 75.700} C_DIS
LIN {X -0.195,Y -585.023,Z 1475.212,A 0.000,B 0.000,C 90.000,E1 74.102} C_DIS
LIN {X -0.149,Y -585.913,Z 1475.203,A 0.000,B 0.000,C 90.000,E1 72.489} C_DIS
LIN {X -0.048,Y -586.990,Z 1475.192,A 0.000,B 0.000,C 90.000,E1 70.604} C_DIS
LIN {X -0.339,Y -587.827,Z 1475.183,A 0.000,B 0.000,C 90.000,E1 69.028} C_DIS
LIN {X -0.224,Y -589.223,Z 1475.170,A 0.000,B 0.000,C 90.000,E1 66.613} C_DIS
LIN {X 0.195,Y -590.196,Z 1475.161,A 0.000,B 0.000,C 90.000,E1 64.973} C_DIS
LIN {X 0.000,Y -591.304,Z 1475.151,A 0.000,B 0.000,C 90.000,E1 63.127} C_DIS
LIN {X -0.007,Y -592.853,Z 1475.139,A 0.000,B 0.000,C 90.000,E1 61.001} C_DIS
LIN {X 0.186,Y -594.385,Z 1475.129,A 0.000,B 0.000,C 90.000,E1 59.125} C_DIS
LIN {X -0.075,Y -595.901,Z 1475.118,A 0.000,B 0.000,C 90.000,E1 57.296} C_DIS
LIN {X 0.168,Y -596.804,Z 1475.112,A 0.000,B 0.000,C 90.000,E1 56.215} C_DIS
LIN {X 0.041,Y -598.102,Z 1475.104,A 0.000,B 0.000,C 90.000,E1 54.642} C_DIS
LIN {X 0.146,Y -599.199,Z 1475.095,A 0.000,B 0.000,C 90.000,E1 53.050} C_DIS
LIN {X 0.042,Y -600.069,Z 1475.088,A 0.000,B 0.000,C 90.000,E1 51.743} C_DIS
LIN {X -0.295,Y -600.655,Z 1475.082,A 0.000,B 0.000,C 90.000,E1 50.723} C_DIS
LIN {X -0.028,Y -601.030,Z 1475.077,A 0.000,B 0.000,C 90.000,E1 49.908} C_DIS
LIN {X 0.241,Y -601.321,Z 1475.073,A 0.000,B 0.000,C 90.000,E1 49.094} C_DIS
LIN {X 0.083,Y -601.524,Z 1475.066,A 0.000,B 0.000,C 90.000,E1 47.796} C_DIS
LIN {X -0.101,Y -601.626,Z 1475.061,A 0.000,B 0.000,C 90.000,E1 47.025} C_DIS
LIN {X -0.283,Y -601.602,Z 1475.054,A 0.000,B 0.000,C 90.000,E1 45.729} C_DIS
LIN {X -0.252,Y -601.282,Z 1475.048,A 0.000,B 0.000,C 90.000,E1 44.676} C_DIS
LIN {X -0.229,Y -600.756,Z 1475.042,A 0.000,B 0.000,C 90.000,E1 43.623} C_DIS
LIN {X 0.220,Y -600.064,Z 1475.036,A 0.000,B 0.000,C 90.000,E1 42.528} C_DIS
LIN {X -0.191,Y -599.075,Z 1475.031,A 0.000,B 0.000,C 90.000,E1 41.515} C_DIS
LIN {X 0.054,Y -598.243,Z 1475.026,A 0.000,B 0.000,C 90.000,E1 40.701} C_DIS
LIN {X -0.163,Y -597.300,Z 1475.022,A 0.000,B 0.000,C 90.000,E1 39.930} C_DIS
LIN {X 0.057,Y -595.428,Z 1475.014,A 0.000,B 0.000,C 90.000,E1 38.588} C_DIS
LIN {X 0.121,Y -593.713,Z 1475.009,A 0.000,B 0.000,C 90.000,E1 37.523} C_DIS
LIN {X 0.169,Y -591.770,Z 1475.003,A 0.000,B 0.000,C 90.000,E1 36.457} C_DIS
LIN {X -0.017,Y -590.126,Z 1474.998,A 0.000,B 0.000,C 90.000,E1 35.678} C_DIS
LIN {X -0.221,Y -588.258,Z 1474.994,A 0.000,B 0.000,C 90.000,E1 34.898} C_DIS
LIN {X 0.039,Y -586.070,Z 1474.989,A 0.000,B 0.000,C 90.000,E1 34.072} C_DIS
LIN {X -0.213,Y -583.639,Z 1474.985,A 0.000,B 0.000,C 90.000,E1 33.293} C_DIS
LIN {X -0.153,Y -580.063,Z 1474.979,A 0.000,B 0.000,C 90.000,E1 32.212} C_DIS
LIN {X -0.141,Y -578.052,Z 1474.976,A 0.000,B 0.000,C 90.000,E1 31.671} C_DIS
LIN {X -0.142,Y -575.808,Z 1474.973,A 0.000,B 0.000,C 90.000,E1 31.131} C_DIS
LIN {X -0.241,Y -572.742,Z 1474.969,A 0.000,B 0.000,C 90.000,E1 30.463} C_DIS
LIN {X 0.124,Y -569.398,Z 1474.965,A 0.000,B 0.000,C 90.000,E1 29.745} C_DIS
LIN {X -0.221,Y -564.401,Z 1474.960,A 0.000,B 0.000,C 90.000,E1 28.821} C_DIS
LIN {X -0.131,Y -558.843,Z 1474.955,A 0.000,B 0.000,C 90.000,E1 27.847} C_DIS
LIN {X -0.006,Y -553.465,Z 1474.950,A 0.000,B 0.000,C 90.000,E1 27.001} C_DIS
LIN {X 0.043,Y -549.655,Z 1474.947,A 0.000,B 0.000,C 90.000,E1 26.437} C_DIS
LIN {X -0.064,Y -542.523,Z 1474.942,A 0.000,B 0.000,C 90.000,E1 25.463} C_DIS
LIN {X 0.043,Y -539.129,Z 1474.939,A 0.000,B 0.000,C 90.000,E1 25.027} C_DIS
LIN {X 0.153,Y -535.239,Z 1474.937,A 0.000,B 0.000,C 90.000,E1 24.591} C_DIS
LIN {X -0.012,Y -532.306,Z 1474.935,A 0.000,B 0.000,C 90.000,E1 24.335} C_DIS
LIN {X 0.001,Y -529.083,Z 1474.934,A 0.000,B 0.000,C 90.000,E1 24.079} C_DIS
LIN {X 0.077,Y -526.309,Z 1474.933,A 0.000,B 0.000,C 90.000,E1 23.898} C_DIS
LIN {X -0.120,Y -524.002,Z 1474.932,A 0.000,B 0.000,C 90.000,E1 23.823} C_DIS
LIN {X 0.063,Y -522.171,Z 1474.932,A 0.000,B 0.000,C 90.000,E1 23.770} C_DIS
LIN {X 0.021,Y -381.150,Z 1474.932,A 0.000,B 0.000,C 90.000,E1 23.770} C_DIS
LIN {X -0.036,Y -375.016,Z 1474.906,A 0.000,B 0.000,C 90.000,E1 19.033} C_DIS
LIN {X -0.118,Y -373.691,Z 1474.898,A 0.000,B 0.000,C 90.000,E1 17.583} C_DIS
LIN {X 0.017,Y -368.087,Z 1474.869,A 0.000,B 0.000,C 90.000,E1 12.411} C_DIS
LIN {X -0.175,Y -366.408,Z 1474.855,A 0.000,B 0.000,C 90.000,E1 9.849} C_DIS
LIN {X 0.124,Y -361.743,Z 1474.822,A 0.000,B 0.000,C 90.000,E1 3.841} C_DIS
LIN {X 0.010,Y -360.865,Z 1474.801,A 0.000,B 0.000,C 90.000,E1 0.115} C_DIS
LIN {X -0.053,Y -359.426,Z 1474.770,A 0.000,B 0.000,C 90.000,E1 354.546} C_DIS
LIN {X 0.070,Y -358.890,Z 1474.759,A 0.000,B 0.000,C 90.000,E1 352.648} C_DIS
LIN {X -0.020,Y -359.563,Z 1474.726,A 0.000,B 0.000,C 90.000,E1 346.645} C_DIS
LIN {X 0.001,Y -361.801,Z 1474.684,A 0.000,B 0.000,C 90.000,E1 339.135} C_DIS
LIN {X -0.154,Y -362.053,Z 1474.680,A 0.000,B 0.000,C 90.000,E1 338.411} C_DIS
LIN {X 0.189,Y -365.980,Z 1474.643,A 0.000,B 0.000,C 90.000,E1 331.641} C_DIS
LIN {X 0.029,Y -366.387,Z 1474.639,A 0.000,B 0.000,C 90.000,E1 330.923} C_DIS
LIN {X -0.031,Y -371.355,Z 1474.604,A 0.000,B 0.000,C 90.000,E1 324.642} C_DIS
LIN {X -0.043,Y -371.766,Z 1474.602,A 0.000,B 0.000,C 90.000,E1 324.276} C_DIS
LIN {X 0.013,Y -377.358,Z 1474.567,A 0.000,B 0.000,C 90.000,E1 318.038} C_DIS
LIN {X 0.012,Y -378.235,Z 1474.563,A 0.000,B 0.000,C 90.000,E1 317.310} C_DIS
LIN {X 0.002,Y -383.940,Z 1474.531,A 0.000,B 0.000,C 90.000,E1 311.515} C_DIS
LIN {X 0.088,Y -384.893,Z 1474.527,A 0.000,B 0.000,C 90.000,E1 310.782} C_DIS
LIN {X 0.262,Y -390.610,Z 1474.495,A 0.000,B 0.000,C 90.000,E1 305.025} C_DIS
LIN {X 0.106,Y -391.104,Z 1474.493,A 0.000,B 0.000,C 90.000,E1 304.692} C_DIS
LIN {X 0.022,Y -391.648,Z 1474.489,A 0.000,B 0.000,C 90.000,E1 303.992} C_DIS
LIN {X -0.080,Y -396.825,Z 1474.459,A 0.000,B 0.000,C 90.000,E1 298.693} C_DIS
LIN {X -0.210,Y -397.120,Z 1474.457,A 0.000,B 0.000,C 90.000,E1 298.359} C_DIS
LIN {X -0.055,Y -401.597,Z 1474.426,A 0.000,B 0.000,C 90.000,E1 292.717} C_DIS
LIN {X 0.222,Y -404.659,Z 1474.395,A 0.000,B 0.000,C 90.000,E1 287.094} C_DIS
LIN {X -0.079,Y -404.735,Z 1474.391,A 0.000,B 0.000,C 90.000,E1 286.441} C_DIS
LIN {X 0.214,Y -406.099,Z 1474.364,A 0.000,B 0.000,C 90.000,E1 281.535} C_DIS
LIN {X -0.176,Y -406.094,Z 1474.362,A 0.000,B 0.000,C 90.000,E1 281.243} C_DIS
LIN {X -0.097,Y -405.680,Z 1474.333,A 0.000,B 0.000,C 90.000,E1 276.024} C_DIS
LIN {X -0.165,Y -405.058,Z 1474.328,A 0.000,B 0.000,C 90.000,E1 274.992} C_DIS
LIN {X -0.060,Y -403.497,Z 1474.304,A 0.000,B 0.000,C 90.000,E1 270.802} C_DIS
LIN {X -0.092,Y -403.288,Z 1474.302,A 0.000,B 0.000,C 90.000,E1 270.458} C_DIS
LIN {X 0.091,Y -398.931,Z 1474.271,A 0.000,B 0.000,C 90.000,E1 264.837} C_DIS
LIN {X -0.040,Y -393.108,Z 1474.242,A 0.000,B 0.000,C 90.000,E1 259.567} C_DIS
LIN {X -0.079,Y -392.835,Z 1474.240,A 0.000,B 0.000,C 90.000,E1 259.218} C_DIS
LIN {X 0.034,Y -385.993,Z 1474.212,A 0.000,B 0.000,C 90.000,E1 254.212} C_DIS
LIN {X -0.026,Y -385.267,Z 1474.208,A 0.000,B 0.000,C 90.000,E1 253.504} C_DIS
LIN {X -0.004,Y -384.768,Z 1474.206,A 0.000,B 0.000,C 90.000,E1 253.142} C_DIS
LIN {X 0.221,Y -377.973,Z 1474.182,A 0.000,B 0.000,C 90.000,E1 248.773} C_DIS
LIN {X -0.044,Y -376.233,Z 1474.174,A 0.000,B 0.000,C 90.000,E1 247.358} C_DIS
LIN {X 0.057,Y -374.944,Z 1474.170,A 0.000,B 0.000,C 90.000,E1 246.613} C_DIS
LIN {X -0.208,Y -368.417,Z 1474.148,A 0.000,B 0.000,C 90.000,E1 242.615} C_DIS
LIN {X 0.097,Y -366.047,Z 1474.137,A 0.000,B 0.000,C 90.000,E1 240.717} C_DIS
LIN {X 0.004,Y -359.196,Z 1474.115,A 0.000,B 0.000,C 90.000,E1 236.628} C_DIS
LIN {X 0.021,Y -355.842,Z 1474.100,A 0.000,B 0.000,C 90.000,E1 233.989} C_DIS
LIN {X -0.173,Y -348.793,Z 1474.075,A 0.000,B 0.000,C 90.000,E1 229.461} C_DIS
LIN {X -0.097,Y -346.185,Z 1474.062,A 0.000,B 0.000,C 90.000,E1 227.148} C_DIS
LIN {X -0.088,Y -345.065,Z 1474.058,A 0.000,B 0.000,C 90.000,E1 226.377} C_DIS
LIN {X 0.094,Y -338.586,Z 1474.030,A 0.000,B 0.000,C 90.000,E1 221.310} C_DIS
LIN {X 0.094,Y -336.840,Z 1474.019,A 0.000,B 0.000,C 90.000,E1 219.358} C_DIS
LIN {X 0.014,Y -330.861,Z 1473.988,A 0.000,B 0.000,C 90.000,E1 213.865} C_DIS
LIN {X 0.149,Y -329.296,Z 1473.975,A 0.000,B 0.000,C 90.000,E1 211.465} C_DIS
LIN {X -0.154,Y -324.669,Z 1473.942,A 0.000,B 0.000,C 90.000,E1 205.540} C_DIS
LIN {X 0.174,Y -323.837,Z 1473.928,A 0.000,B 0.000,C 90.000,E1 203.078} C_DIS
LIN {X -0.017,Y -321.124,Z 1473.881,A 0.000,B 0.000,C 90.000,E1 194.662} C_DIS
LIN {X 0.138,Y -320.932,Z 1473.877,A 0.000,B 0.000,C 90.000,E1 193.828} C_DIS
LIN {X -0.076,Y -321.562,Z 1473.832,A 0.000,B 0.000,C 90.000,E1 185.796} C_DIS
LIN {X -0.143,Y -324.415,Z 1473.790,A 0.000,B 0.000,C 90.000,E1 178.165} C_DIS
LIN {X -0.141,Y -325.376,Z 1473.783,A 0.000,B 0.000,C 90.000,E1 176.963} C_DIS
LIN {X -0.100,Y -329.112,Z 1473.750,A 0.000,B 0.000,C 90.000,E1 170.971} C_DIS
LIN {X 0.061,Y -334.260,Z 1473.726,A 0.000,B 0.000,C 90.000,E1 166.589} C_DIS
LIN {X 0.067,Y -335.488,Z 1473.719,A 0.000,B 0.000,C 90.000,E1 165.408} C_DIS
LIN {X 0.143,Y -340.932,Z 1473.695,A 0.000,B 0.000,C 90.000,E1 161.094} C_DIS
LIN {X -0.172,Y -342.138,Z 1473.691,A 0.000,B 0.000,C 90.000,E1 160.369} C_DIS
LIN {X -0.058,Y -347.939,Z 1473.667,A 0.000,B 0.000,C 90.000,E1 156.102} C_DIS
LIN {X 0.015,Y -350.374,Z 1473.659,A 0.000,B 0.000,C 90.000,E1 154.665} C_DIS
LIN {X -0.027,Y -482.727,Z 1473.659,A 0.000,B 0.000,C 90.000,E1 154.665} C_DIS
LIN {X 0.188,Y -486.514,Z 1473.659,A 0.000,B 0.000,C 90.000,E1 154.537} C_DIS
LIN {X -0.059,Y -488.738,Z 1473.658,A 0.000,B 0.000,C 90.000,E1 154.460} C_DIS
LIN {X 0.092,Y -491.526,Z 1473.657,A 0.000,B 0.000,C 90.000,E1 154.280} C_DIS
LIN {X 0.135,Y -495.717,Z 1473.656,A 0.000,B 0.000,C 90.000,E1 153.973} C_DIS
LIN {X -0.103,Y -498.547,Z 1473.654,A 0.000,B 0.000,C 90.000,E1 153.768} C_DIS
LIN {X -0.134,Y -502.592,Z 1473.652,A 0.000,B 0.000,C 90.000,E1 153.384} C_DIS
LIN {X 0.005,Y -507.630,Z 1473.649,A 0.000,B 0.000,C 90.000,E1 152.794} C_DIS
LIN {X -0.268,Y -512.359,Z 1473.646,A 0.000,B 0.000,C 90.000,E1 152.231} C_DIS
LIN {X 0.003,Y -517.595,Z 1473.641,A 0.000,B 0.000,C 90.000,E1 151.463} C_DIS
LIN {X 0.031,Y -521.260,Z 1473.638,A 0.000,B 0.000,C 90.000,E1 150.873} C_DIS
LIN {X 0.086,Y -524.521,Z 1473.635,A 0.000,B 0.000,C 90.000,E1 150.284} C_DIS
LIN {X 0.118,Y -528.791,Z 1473.630,A 0.000,B 0.000,C 90.000,E1 149.410} C_DIS
LIN {X -0.074,Y -530.818,Z 1473.628,A 0.000,B 0.000,C 90.000,E1 148.997} C_DIS
LIN {X 0.048,Y -533.163,Z 1473.625,A 0.000,B 0.000,C 90.000,E1 148.408} C_DIS
LIN {X 0.171,Y -536.190,Z 1473.620,A 0.000,B 0.000,C 90.000,E1 147.533} C_DIS
LIN {X -0.125,Y -539.002,Z 1473.615,A 0.000,B 0.000,C 90.000,E1 146.707} C_DIS
LIN {X -0.105,Y -540.709,Z 1473.612,A 0.000,B 0.000,C 90.000,E1 146.135} C_DIS
LIN {X 0.122,Y -543.832,Z 1473.606,A 0.000,B 0.000,C 90.000,E1 144.975} C_DIS
LIN {X 0.222,Y -545.912,Z 1473.601,A 0.000,B 0.000,C 90.000,E1 144.116} C_DIS
LIN {X 0.021,Y -547.716,Z 1473.596,A 0.000,B 0.000,C 90.000,E1 143.290} C_DIS
LIN {X -0.223,Y -549.840,Z 1473.590,A 0.000,B 0.000,C 90.000,E1 142.190} C_DIS
LIN {X -0.003,Y -551.607,Z 1473.584,A 0.000,B 0.000,C 90.000,E1 141.045} C_DIS
LIN {X 0.159,Y -553.138,Z 1473.577,A 0.000,B 0.000,C 90.000,E1 139.908} C_DIS
LIN {X -0.076,Y -554.214,Z 1473.573,A 0.000,B 0.000,C 90.000,E1 139.094} C_DIS
LIN {X 0.125,Y -555.450,Z 1473.567,A 0.000,B 0.000,C 90.000,E1 137.957} C_DIS
LIN {X -0.031,Y -556.847,Z 1473.559,A 0.000,B 0.000,C 90.000,E1 136.581} C_DIS
LIN {X -0.201,Y -557.815,Z 1473.553,A 0.000,B 0.000,C 90.000,E1 135.486} C_DIS
LIN {X 0.148,Y -559.137,Z 1473.543,A 0.000,B 0.000,C 90.000,E1 133.785} C_DIS
LIN {X 0.087,Y -559.876,Z 1473.536,A 0.000,B 0.000,C 90.000,E1 132.405} C_DIS
LIN {X -0.041,Y -560.347,Z 1473.530,A 0.000,B 0.000,C 90.000,E1 131.310} C_DIS
LIN {X 0.255,Y -560.644,Z 1473.523,A 0.000,B 0.000,C 90.000,E1 130.172} C_DIS
LIN {X -0.051,Y -560.846,Z 1473.514,A 0.000,B 0.000,C 90.000,E1 128.543} C_DIS
LIN {X 0.180,Y -561.043,Z 1473.503,A 0.000,B 0.000,C 90.000,E1 126.583} C_DIS
LIN {X -0.313,Y -561.078,Z 1473.499,A 0.000,B 0.000,C 90.000,E1 125.804} C_DIS
LIN {X -0.252,Y -560.861,Z 1473.493,A 0.000,B 0.000,C 90.000,E1 124.692} C_DIS
LIN {X 0.287,Y -560.456,Z 1473.476,A 0.000,B 0.000,C 90.000,E1 121.592} C_DIS
LIN {X -0.033,Y -560.597,Z 1473.463,A 0.000,B 0.000,C 90.000,E1 119.411} C_DIS
LIN {X -0.215,Y -560.861,Z 1473.454,A 0.000,B 0.000,C 90.000,E1 117.769} C_DIS
LIN {X 0.146,Y -561.231,Z 1473.443,A 0.000,B 0.000,C 90.000,E1 115.796} C_DIS
LIN {X -0.024,Y -561.666,Z 1473.434,A 0.000,B 0.000,C 90.000,E1 114.155} C_DIS
LIN {X 0.209,Y -562.074,Z 1473.428,A 0.000,B 0.000,C 90.000,E1 113.025} C_DIS
LIN {X 0.143,Y -562.666,Z 1473.417,A 0.000,B 0.000,C 90.000,E1 111.099} C_DIS
LIN {X -0.318,Y -563.141,Z 1473.407,A 0.000,B 0.000,C 90.000,E1 109.214} C_DIS
LIN {X -0.156,Y -563.487,Z 1473.399,A 0.000,B 0.000,C 90.000,E1 107.819} C_DIS
LIN {X -0.243,Y -564.033,Z 1473.388,A 0.000,B 0.000,C 90.000,E1 105.898} C_DIS
LIN {X 0.063,Y -564.669,Z 1473.378,A 0.000,B 0.000,C 90.000,E1 103.939} C_DIS
LIN {X -0.264,Y -565.531,Z 1473.365,A 0.000,B 0.000,C 90.000,E1 101.771} C_DIS
LIN {X -0.285,Y -566.334,Z 1473.355,A 0.000,B 0.000,C 90.000,E1 99.849} C_DIS
LIN {X 0.095,Y -567.082,Z 1473.345,A 0.000,B 0.000,C 90.000,E1 98.163} C_DIS
LIN {X 0.106,Y -568.211,Z 1473.333,A 0.000,B 0.000,C 90.000,E1 95.967} C_DIS
LIN {X -0.247,Y -569.233,Z 1473.324,A 0.000,B 0.000,C 90.000,E1 94.359} C_DIS
LIN {X -0.006,Y -570.388,Z 1473.315,A 0.000,B 0.000,C 90.000,E1 92.694} C_DIS
LIN {X 0.095,Y -571.398,Z 1473.307,A 0.000,B 0.000,C 90.000,E1 91.318} C_DIS
LIN {X 0.048,Y -573.068,Z 1473.295,A 0.000,B 0.000,C 90.000,E1 89.141} C_DIS
LIN {X 0.201,Y -574.079,Z 1473.288,A 0.000,B 0.000,C 90.000,E1 87.764} C_DIS
LIN {X -0.058,Y -575.366,Z 1473.279,A 0.000,B 0.000,C 90.000,E1 86.159} C_DIS
LIN {X -0.211,Y -576.644,Z 1473.270,A 0.000,B 0.000,C 90.000,E1 84.546} C_DIS
LIN {X 0.023,Y -578.492,Z 1473.258,A 0.000,B 0.000,C 90.000,E1 82.356} C_DIS
LIN {X -0.114,Y -580.328,Z 1473.246,A 0.000,B 0.000,C 90.000,E1 80.208} C_DIS
LIN {X 0.121,Y -581.261,Z 1473.240,A 0.000,B 0.000,C 90.000,E1 79.106} C_DIS
LIN {X 0.039,Y -582.931,Z 1473.229,A 0.000,B 0.000,C 90.000,E1 77.229} C_DIS
LIN {X 0.084,Y -584.071,Z 1473.222,A 0.000,B 0.000,C 90.000,E1 75.880} C_DIS
LIN {X -0.190,Y -584.563,Z 1473.217,A 0.000,B 0.000,C 90.000,E1 75.102} C_DIS
LIN {X 0.022,Y -585.430,Z 1473.210,A 0.000,B 0.000,C 90.000,E1 73.740} C_DIS
LIN {X -0.070,Y -586.427,Z 1473.199,A 0.000,B 0.000,C 90.000,E1 71.873} C_DIS
LIN {X -0.228,Y -587.194,Z 1473.192,A 0.000,B 0.000,C 90.000,E1 70.550} C_DIS
LIN {X -0.185,Y -587.942,Z 1473.184,A 0.000,B 0.000,C 90.000,E1 69.209} C_DIS
LIN {X -0.061,Y -589.297,Z 1473.171,A 0.000,B 0.000,C 90.000,E1 66.794} C_DIS
LIN {X 0.009,Y -590.442,Z 1473.161,A 0.000,B 0.000,C 90.000,E1 64.921} C_DIS
LIN {X 0.078,Y -591.563,Z 1473.150,A 0.000,B 0.000,C 90.000,E1 63.050} C_DIS
LIN {X -0.012,Y -593.333,Z 1473.137,A 0.000,B 0.000,C 90.000,E1 60.667} C_DIS
LIN {X 0.198,Y -594.910,Z 1473.127,A 0.000,B 0.000,C 90.000,E1 58.791} C_DIS
LIN {X -0.155,Y -596.695,Z 1473.115,A 0.000,B 0.000,C 90.000,E1 56.707} C_DIS
LIN {X -0.176,Y -597.731,Z 1473.108,A 0.000,B 0.000,C 90.000,E1 55.388} C_DIS
LIN {X -0.069,Y -598.577,Z 1473.102,A 0.000,B 0.000,C 90.000,E1 54.322} C_DIS
LIN {X 0.176,Y -599.651,Z 1473.093,A 0.000,B 0.000,C 90.000,E1 52.718} C_DIS
LIN {X -0.155,Y -600.713,Z 1473.084,A 0.000,B 0.000,C 90.000,E1 51.170} C_DIS
LIN {X -0.104,Y -601.244,Z 1473.078,A 0.000,B 0.000,C 90.000,E1 50.114} C_DIS
LIN {X -0.041,Y -601.593,Z 1473.073,A 0.000,B 0.000,C 90.000,E1 49.057} C_DIS
LIN {X 0.053,Y -601.859,Z 1473.064,A 0.000,B 0.000,C 90.000,E1 47.472} C_DIS
LIN {X 0.314,Y -601.922,Z 1473.057,A 0.000,B 0.000,C 90.000,E1 46.134} C_DIS
LIN {X -0.299,Y -601.857,Z 1473.052,A 0.000,B 0.000,C 90.000,E1 45.405} C_DIS
LIN {X 0.380,Y -601.325,Z 1473.045,A 0.000,B 0.000,C 90.000,E1 44.028} C_DIS
LIN {X -0.221,Y -600.514,Z 1473.038,A 0.000,B 0.000,C 90.000,E1 42.771} C_DIS
LIN {X -0.008,Y -599.859,Z 1473.033,A 0.000,B 0.000,C 90.000,E1 41.962} C_DIS
LIN {X 0.255,Y -598.474,Z 1473.026,A 0.000,B 0.000,C 90.000,E1 40.620} C_DIS
LIN {X 0.271,Y -597.179,Z 1473.020,A 0.000,B 0.000,C 90.000,E1 39.564} C_DIS
LIN {X -0.110,Y -595.633,Z 1473.014,A 0.000,B 0.000,C 90.000,E1 38.543} C_DIS
LIN {X 0.325,Y -593.939,Z 1473.008,A 0.000,B 0.000,C 90.000,E1 37.443} C_DIS
LIN {X -0.103,Y -592.015,Z 1473.002,A 0.000,B 0.000,C 90.000,E1 36.423} C_DIS
LIN {X -0.086,Y -589.748,Z 1472.996,A 0.000,B 0.000,C 90.000,E1 35.358} C_DIS
LIN {X -0.017,Y -588.478,Z 1472.994,A 0.000,B 0.000,C 90.000,E1 34.818} C_DIS
LIN {X 0.242,Y -586.266,Z 1472.989,A 0.000,B 0.000,C 90.000,E1 33.992} C_DIS
LIN {X -0.011,Y -583.826,Z 1472.985,A 0.000,B 0.000,C 90.000,E1 33.214} C_DIS
LIN {X -0.119,Y -581.223,Z 1472.980,A 0.000,B 0.000,C 90.000,E1 32.418} C_DIS
LIN {X 0.059,Y -578.284,Z 1472.976,A 0.000,B 0.000,C 90.000,E1 31.592} C_DIS
LIN {X -0.099,Y -574.820,Z 1472.971,A 0.000,B 0.000,C 90.000,E1 30.797} C_DIS
LIN {X -0.125,Y -572.331,Z 1472.968,A 0.000,B 0.000,C 90.000,E1 30.256} C_DIS
LIN {X 0.319,Y -569.626,Z 1472.965,A 0.000,B 0.000,C 90.000,E1 29.667} C_DIS
LIN {X -0.028,Y -564.627,Z 1472.960,A 0.000,B 0.000,C 90.000,E1 28.743} C_DIS
LIN {X 0.059,Y -559.059,Z 1472.954,A 0.000,B 0.000,C 90.000,E1 27.769} C_DIS
LIN {X -0.070,Y -553.693,Z 1472.950,A 0.000,B 0.000,C 90.000,E1 26.950} C_DIS
LIN {X 0.228,Y -549.925,Z 1472.947,A 0.000,B 0.000,C 90.000,E1 26.360} C_DIS
LIN {X -0.114,Y -542.807,Z 1472.941,A 0.000,B 0.000,C 90.000,E1 25.412} C_DIS
LIN {X -0.042,Y -537.245,Z 1472.937,A 0.000,B 0.000,C 90.000,E1 24.695} C_DIS
LIN {X 0.034,Y -533.521,Z 1472.935,A 0.000,B 0.000,C 90.000,E1 24.259} C_DIS
LIN {X 0.195,Y -529.286,Z 1472.932,A 0.000,B 0.000,C 90.000,E1 23.823} C_DIS
LIN {X -0.061,Y -526.137,Z 1472.931,A 0.000,B 0.000,C 90.000,E1 23.590} C_DIS
LIN {X 0.027,Y -524.491,Z 1472.930,A 0.000,B 0.000,C 90.000,E1 23.462} C_DIS
LIN {X -0.323,Y -521.460,Z 1472.929,A 0.000,B 0.000,C 90.000,E1 23.334} C_DIS
LIN {X 0.121,Y -519.139,Z 1472.929,A 0.000,B 0.000,C 90.000,E1 23.206} C_DIS
LIN {X -0.008,Y -518.127,Z 1472.929,A 0.000,B 0.000,C 90.000,E1 23.206} C_DIS
LIN {X -0.029,Y -380.258,Z 1472.929,A 0.000,B 0.000,C 90.000,E1 23.206} C_DIS
LIN {X 0.043,Y -374.112,Z 1472.900,A 0.000,B 0.000,C 90.000,E1 18.055} C_DIS
LIN {X -0.007,Y -373.424,Z 1472.896,A 0.000,B 0.000,C 90.000,E1 17.330} C_DIS
LIN {X 0.004,Y -367.902,Z 1472.868,A 0.000,B 0.000,C 90.000,E1 12.175} C_DIS
LIN {X -0.053,Y -366.501,Z 1472.855,A 0.000,B 0.000,C 90.000,E1 9.962} C_DIS
LIN {X -0.118,Y -361.801,Z 1472.822,A 0.000,B 0.000,C 90.000,E1 4.012} C_DIS
LIN {X 0.128,Y -360.903,Z 1472.801,A 0.000,B 0.000,C 90.000,E1 0.229} C_DIS
LIN {X -0.053,Y -359.426,Z 1472.770,A 0.000,B 0.000,C 90.000,E1 354.546} C_DIS
LIN {X 0.070,Y -358.890,Z 1472.759,A 0.000,B 0.000,C 90.000,E1 352.648} C_DIS
LIN {X -0.020,Y -359.563,Z 1472.726,A 0.000,B 0.000,C 90.000,E1 346.645} C_DIS
LIN {X 0.001,Y -361.801,Z 1472.684,A 0.000,B 0.000,C 90.000,E1 339.135} C_DIS
LIN {X -0.154,Y -362.053,Z 1472.680,A 0.000,B 0.000,C 90.000,E1 338.411} C_DIS
LIN {X 0.189,Y -365.980,Z 1472.643,A 0.000,B 0.000,C 90.000,E1 331.641} C_DIS
LIN {X 0.029,Y -366.387,Z 1472.639,A 0.000,B 0.000,C 90.000,E1 330.923} C_DIS
LIN {X -0.031,Y -371.355,Z 1472.604,A 0.000,B 0.000,C 90.000,E1 324.642} C_DIS
LIN {X -0.043,Y -371.766,Z 1472.602,A 0.000,B 0.000,C 90.000,E1 324.276} C_DIS
LIN {X 0.013,Y -377.358,Z 1472.567,A 0.000,B 0.000,C 90.000,E1 318.038} C_DIS
LIN {X 0.012,Y -378.235,Z 1472.563,A 0.000,B 0.000,C 90.000,E1 317.310} C_DIS
LIN {X 0.002,Y -383.940,Z 1472.531,A 0.000,B 0.000,C 90.000,E1 311.515} C_DIS
LIN {X 0.088,Y -384.893,Z 1472.527,A 0.000,B 0.000,C 90.000,E1 310.782} C_DIS
LIN {X 0.262,Y -390.610,Z 1472.495,A 0.000,B 0.000,C 90.000,E1 305.025} C_DIS
LIN {X 0.106,Y -391.104,Z 1472.493,A 0.000,B 0.000,C 90.000,E1 304.692} C_DIS
LIN {X 0.022,Y -391.648,Z 1472.489,A 0.000,B 0.000,C 90.000,E1 303.992} C_DIS
LIN {X -0.080,Y -396.825,Z 1472.459,A 0.000,B 0.000,C 90.000,E1 298.693} C_DIS
LIN {X -0.210,Y -397.120,Z 1472.457,A 0.000,B 0.000,C 90.000,E1 298.359} C_DIS
LIN {X -0.055,Y -401.597,Z 1472.426,A 0.000,B 0.000,C 90.000,E1 292.717} C_DIS
LIN {X 0.222,Y -404.659,Z 1472.395,A 0.000,B 0.000,C 90.000,E1 287.094} C_DIS
LIN {X -0.079,Y -404.735,Z 1472.391,A 0.000,B 0.000,C 90.000,E1 286.441} C_DIS
LIN {X 0.214,Y -406.099,Z 1472.364,A 0.000,B 0.000,C 90.000,E1 281.535} C_DIS
LIN {X -0.176,Y -406.094,Z 1472.362,A 0.000,B 0.000,C 90.000,E1 281.243} C_DIS
LIN {X -0.097,Y -405.680,Z 1472.333,A 0.000,B 0.000,C 90.000,E1 276.024} C_DIS
LIN {X -0.165,Y -405.058,Z 1472.328,A 0.000,B 0.000,C 90.000,E1 274.992} C_DIS
LIN {X -0.060,Y -403.497,Z 1472.304,A 0.000,B 0.000,C 90.000,E1 270.802} C_DIS
LIN {X -0.092,Y -403.288,Z 1472.302,A 0.000,B 0.000,C 90.000,E1 270.458} C_DIS
LIN {X 0.091,Y -398.931,Z 1472.271,A 0.000,B 0.000,C 90.000,E1 264.837} C_DIS
LIN {X -0.040,Y -393.108,Z 1472.242,A 0.000,B 0.000,C 90.000,E1 259.567} C_DIS
LIN {X -0.079,Y -392.835,Z 1472.240,A 0.000,B 0.000,C 90.000,E1 259.218} C_DIS
LIN {X 0.034,Y -385.993,Z 1472.212,A 0.000,B 0.000,C 90.000,E1 254.212} C_DIS
LIN {X -0.026,Y -385.267,Z 1472.208,A 0.000,B 0.000,C 90.000,E1 253.504} C_DIS
LIN {X -0.004,Y -384.768,Z 1472.206,A 0.000,B 0.000,C 90.000,E1 253.142} C_DIS
LIN {X 0.221,Y -377.973,Z 1472.182,A 0.000,B 0.000,C 90.000,E1 248.773} C_DIS
LIN {X -0.044,Y -376.233,Z 1472.174,A 0.000,B 0.000,C 90.000,E1 247.358} C_DIS
LIN {X 0.057,Y -374.944,Z 1472.170,A 0.000,B 0.000,C 90.000,E1 246.613} C_DIS
LIN {X -0.208,Y -368.417,Z 1472.148,A 0.000,B 0.000,C 90.000,E1 242.615} C_DIS
LIN {X 0.097,Y -366.047,Z 1472.137,A 0.000,B 0.000,C 90.000,E1 240.717} C_DIS
LIN {X 0.004,Y -359.196,Z 1472.115,A 0.000,B 0.000,C 90.000,E1 236.628} C_DIS
LIN {X 0.021,Y -355.842,Z 1472.100,A 0.000,B 0.000,C 90.000,E1 233.989} C_DIS
LIN {X -0.173,Y -348.793,Z 1472.075,A 0.000,B 0.000,C 90.000,E1 229.461} C_DIS
LIN {X -0.097,Y -346.185,Z 1472.062,A 0.000,B 0.000,C 90.000,E1 227.148} C_DIS
LIN {X -0.088,Y -345.065,Z 1472.058,A 0.000,B 0.000,C 90.000,E1 226.377} C_DIS
LIN {X 0.094,Y -338.586,Z 1472.030,A 0.000,B 0.000,C 90.000,E1 221.310} C_DIS
LIN {X 0.094,Y -336.840,Z 1472.019,A 0.000,B 0.000,C 90.000,E1 219.358} C_DIS
LIN {X 0.014,Y -330.861,Z 1471.988,A 0.000,B 0.000,C 90.000,E1 213.865} C_DIS
LIN {X 0.149,Y -329.296,Z 1471.975,A 0.000,B 0.000,C 90.000,E1 211.465} C_DIS
LIN {X -0.154,Y -324.669,Z 1471.942,A 0.000,B 0.000,C 90.000,E1 205.540} C_DIS
LIN {X 0.174,Y -323.837,Z 1471.928,A 0.000,B 0.000,C 90.000,E1 203.078} C_DIS
LIN {X -0.017,Y -321.124,Z 1471.881,A 0.000,B 0.000,C 90.000,E1 194.662} C_DIS
LIN {X 0.138,Y -320.932,Z 1471.877,A 0.000,B 0.000,C 90.000,E1 193.828} C_DIS
LIN {X -0.076,Y -321.562,Z 1471.832,A 0.000,B 0.000,C 90.000,E1 185.796} C_DIS
LIN {X -0.143,Y -324.415,Z 1471.790,A 0.000,B 0.000,C 90.000,E1 178.165} C_DIS
LIN {X -0.141,Y -325.376,Z 1471.783,A 0.000,B 0.000,C 90.000,E1 176.963} C_DIS
LIN {X -0.100,Y -329.112,Z 1471.750,A 0.000,B 0.000,C 90.000,E1 170.971} C_DIS
LIN {X 0.061,Y -334.260,Z 1471.726,A 0.000,B 0.000,C 90.000,E1 166.589} C_DIS
LIN {X 0.067,Y -335.488,Z 1471.719,A 0.000,B 0.000,C 90.000,E1 165.408} C_DIS
LIN {X 0.143,Y -340.932,Z 1471.695,A 0.000,B 0.000,C 90.000,E1 161.094} C_DIS
LIN {X -0.172,Y -342.138,Z 1471.691,A 0.000,B 0.000,C 90.000,E1 160.369} C_DIS
LIN {X -0.058,Y -347.939,Z 1471.667,A 0.000,B 0.000,C 90.000,E1 156.102} C_DIS
LIN {X -0.058,Y -349.400,Z 1471.662,A 0.000,B 0.000,C 90.000,E1 155.229} C_DIS
LIN {X -0.123,Y -476.979,Z 1471.662,A 0.000,B 0.000,C 90.000,E1 155.229} C_DIS
LIN {X -0.211,Y -478.015,Z 1471.662,A 0.000,B 0.000,C 90.000,E1 155.229} C_DIS
LIN {X -0.125,Y -480.540,Z 1471.662,A 0.000,B 0.000,C 90.000,E1 155.153} C_DIS
LIN {X -0.238,Y -482.172,Z 1471.662,A 0.000,B 0.000,C 90.000,E1 155.101} C_DIS
LIN {X 0.174,Y -484.824,Z 1471.661,A 0.000,B 0.000,C 90.000,E1 154.921} C_DIS
LIN {X -0.167,Y -487.639,Z 1471.660,A 0.000,B 0.000,C 90.000,E1 154.793} C_DIS
LIN {X 0.035,Y -491.863,Z 1471.658,A 0.000,B 0.000,C 90.000,E1 154.460} C_DIS
LIN {X 0.061,Y -496.024,Z 1471.656,A 0.000,B 0.000,C 90.000,E1 154.101} C_DIS
LIN {X -0.057,Y -500.114,Z 1471.654,A 0.000,B 0.000,C 90.000,E1 153.717} C_DIS
LIN {X 0.156,Y -505.300,Z 1471.651,A 0.000,B 0.000,C 90.000,E1 153.127} C_DIS
LIN {X 0.085,Y -509.086,Z 1471.648,A 0.000,B 0.000,C 90.000,E1 152.692} C_DIS
LIN {X 0.049,Y -513.706,Z 1471.645,A 0.000,B 0.000,C 90.000,E1 152.103} C_DIS
LIN {X 0.050,Y -517.822,Z 1471.642,A 0.000,B 0.000,C 90.000,E1 151.513} C_DIS
LIN {X 0.082,Y -521.488,Z 1471.639,A 0.000,B 0.000,C 90.000,E1 150.923} C_DIS
LIN {X -0.018,Y -525.477,Z 1471.635,A 0.000,B 0.000,C 90.000,E1 150.205} C_DIS
LIN {X 0.028,Y -529.730,Z 1471.630,A 0.000,B 0.000,C 90.000,E1 149.331} C_DIS
LIN {X 0.297,Y -531.607,Z 1471.627,A 0.000,B 0.000,C 90.000,E1 148.869} C_DIS
LIN {X -0.028,Y -533.917,Z 1471.624,A 0.000,B 0.000,C 90.000,E1 148.329} C_DIS
LIN {X 0.105,Y -536.926,Z 1471.619,A 0.000,B 0.000,C 90.000,E1 147.454} C_DIS
LIN {X -0.182,Y -539.706,Z 1471.615,A 0.000,B 0.000,C 90.000,E1 146.628} C_DIS
LIN {X 0.009,Y -542.182,Z 1471.610,A 0.000,B 0.000,C 90.000,E1 145.754} C_DIS
LIN {X 0.117,Y -545.150,Z 1471.604,A 0.000,B 0.000,C 90.000,E1 144.609} C_DIS
LIN {X -0.088,Y -547.098,Z 1471.599,A 0.000,B 0.000,C 90.000,E1 143.783} C_DIS
LIN {X 0.095,Y -549.300,Z 1471.593,A 0.000,B 0.000,C 90.000,E1 142.637} C_DIS
LIN {X -0.181,Y -550.756,Z 1471.588,A 0.000,B 0.000,C 90.000,E1 141.823} C_DIS
LIN {X 0.051,Y -552.437,Z 1471.582,A 0.000,B 0.000,C 90.000,E1 140.678} C_DIS
LIN {X -0.131,Y -554.241,Z 1471.574,A 0.000,B 0.000,C 90.000,E1 139.299} C_DIS
LIN {X 0.139,Y -555.773,Z 1471.566,A 0.000,B 0.000,C 90.000,E1 137.877} C_DIS
LIN {X -0.010,Y -557.129,Z 1471.558,A 0.000,B 0.000,C 90.000,E1 136.500} C_DIS
LIN {X -0.176,Y -558.081,Z 1471.552,A 0.000,B 0.000,C 90.000,E1 135.405} C_DIS
LIN {X 0.178,Y -559.364,Z 1471.543,A 0.000,B 0.000,C 90.000,E1 133.704} C_DIS
LIN {X 0.120,Y -560.025,Z 1471.535,A 0.000,B 0.000,C 90.000,E1 132.324} C_DIS
LIN {X -0.006,Y -560.492,Z 1471.529,A 0.000,B 0.000,C 90.000,E1 131.229} C_DIS
LIN {X 0.291,Y -560.745,Z 1471.523,A 0.000,B 0.000,C 90.000,E1 130.092} C_DIS
LIN {X 0.080,Y -560.910,Z 1471.512,A 0.000,B 0.000,C 90.000,E1 128.177} C_DIS
LIN {X -0.023,Y -561.148,Z 1471.501,A 0.000,B 0.000,C 90.000,E1 126.251} C_DIS
LIN {X -0.091,Y -561.022,Z 1471.495,A 0.000,B 0.000,C 90.000,E1 125.152} C_DIS
LIN {X -0.205,Y -560.484,Z 1471.481,A 0.000,B 0.000,C 90.000,E1 122.673} C_DIS
LIN {X -0.034,Y -560.461,Z 1471.471,A 0.000,B 0.000,C 90.000,E1 120.718} C_DIS
LIN {X 0.066,Y -560.696,Z 1471.460,A 0.000,B 0.000,C 90.000,E1 118.771} C_DIS
LIN {X -0.113,Y -560.970,Z 1471.451,A 0.000,B 0.000,C 90.000,E1 117.129} C_DIS
LIN {X 0.055,Y -561.474,Z 1471.438,A 0.000,B 0.000,C 90.000,E1 114.899} C_DIS
LIN {X 0.195,Y -562.112,Z 1471.428,A 0.000,B 0.000,C 90.000,E1 112.950} C_DIS
LIN {X -0.083,Y -562.701,Z 1471.417,A 0.000,B 0.000,C 90.000,E1 111.046} C_DIS
LIN {X 0.181,Y -563.197,Z 1471.406,A 0.000,B 0.000,C 90.000,E1 109.087} C_DIS
LIN {X 0.340,Y -563.531,Z 1471.399,A 0.000,B 0.000,C 90.000,E1 107.692} C_DIS
LIN {X 0.093,Y -564.085,Z 1471.388,A 0.000,B 0.000,C 90.000,E1 105.788} C_DIS
LIN {X -0.137,Y -564.728,Z 1471.377,A 0.000,B 0.000,C 90.000,E1 103.883} C_DIS
LIN {X 0.097,Y -565.595,Z 1471.365,A 0.000,B 0.000,C 90.000,E1 101.658} C_DIS
LIN {X -0.302,Y -566.558,Z 1471.353,A 0.000,B 0.000,C 90.000,E1 99.500} C_DIS
LIN {X 0.175,Y -567.392,Z 1471.342,A 0.000,B 0.000,C 90.000,E1 97.530} C_DIS
LIN {X 0.199,Y -568.627,Z 1471.330,A 0.000,B 0.000,C 90.000,E1 95.334} C_DIS
LIN {X -0.145,Y -569.734,Z 1471.321,A 0.000,B 0.000,C 90.000,E1 93.726} C_DIS
LIN {X 0.228,Y -571.112,Z 1471.310,A 0.000,B 0.000,C 90.000,E1 91.776} C_DIS
LIN {X 0.171,Y -572.769,Z 1471.298,A 0.000,B 0.000,C 90.000,E1 89.599} C_DIS
LIN {X -0.272,Y -573.848,Z 1471.290,A 0.000,B 0.000,C 90.000,E1 88.282} C_DIS
LIN {X 0.206,Y -575.318,Z 1471.280,A 0.000,B 0.000,C 90.000,E1 86.331} C_DIS
LIN {X 0.003,Y -576.619,Z 1471.271,A 0.000,B 0.000,C 90.000,E1 84.723} C_DIS
LIN {X 0.222,Y -578.450,Z 1471.259,A 0.000,B 0.000,C 90.000,E1 82.534} C_DIS
LIN {X -0.150,Y -580.085,Z 1471.248,A 0.000,B 0.000,C 90.000,E1 80.679} C_DIS
LIN {X -0.038,Y -581.520,Z 1471.239,A 0.000,B 0.000,C 90.000,E1 79.050} C_DIS
LIN {X 0.118,Y -583.432,Z 1471.227,A 0.000,B 0.000,C 90.000,E1 76.881} C_DIS
LIN {X -0.073,Y -584.313,Z 1471.221,A 0.000,B 0.000,C 90.000,E1 75.825} C_DIS
LIN {X 0.127,Y -585.159,Z 1471.214,A 0.000,B 0.000,C 90.000,E1 74.464} C_DIS
LIN {X 0.267,Y -585.772,Z 1471.208,A 0.000,B 0.000,C 90.000,E1 73.378} C_DIS
LIN {X -0.226,Y -586.647,Z 1471.199,A 0.000,B 0.000,C 90.000,E1 71.819} C_DIS
LIN {X -0.189,Y -587.427,Z 1471.192,A 0.000,B 0.000,C 90.000,E1 70.477} C_DIS
LIN {X -0.133,Y -588.158,Z 1471.184,A 0.000,B 0.000,C 90.000,E1 69.135} C_DIS
LIN {X -0.221,Y -589.501,Z 1471.171,A 0.000,B 0.000,C 90.000,E1 66.741} C_DIS
LIN {X 0.095,Y -590.647,Z 1471.160,A 0.000,B 0.000,C 90.000,E1 64.845} C_DIS
LIN {X 0.012,Y -591.652,Z 1471.151,A 0.000,B 0.000,C 90.000,E1 63.256} C_DIS
LIN {X 0.206,Y -593.371,Z 1471.138,A 0.000,B 0.000,C 90.000,E1 60.845} C_DIS
LIN {X 0.121,Y -594.959,Z 1471.128,A 0.000,B 0.000,C 90.000,E1 58.997} C_DIS
LIN {X -0.131,Y -596.477,Z 1471.118,A 0.000,B 0.000,C 90.000,E1 57.168} C_DIS
LIN {X -0.111,Y -597.196,Z 1471.113,A 0.000,B 0.000,C 90.000,E1 56.373} C_DIS
LIN {X -0.127,Y -598.225,Z 1471.106,A 0.000,B 0.000,C 90.000,E1 55.055} C_DIS
LIN {X -0.016,Y -599.044,Z 1471.100,A 0.000,B 0.000,C 90.000,E1 53.989} C_DIS
LIN {X 0.116,Y -600.112,Z 1471.091,A 0.000,B 0.000,C 90.000,E1 52.396} C_DIS
LIN {X 0.028,Y -601.014,Z 1471.084,A 0.000,B 0.000,C 90.000,E1 51.090} C_DIS
LIN {X -0.302,Y -601.531,Z 1471.078,A 0.000,B 0.000,C 90.000,E1 50.070} C_DIS
LIN {X -0.242,Y -601.845,Z 1471.072,A 0.000,B 0.000,C 90.000,E1 49.013} C_DIS
LIN {X 0.254,Y -602.137,Z 1471.063,A 0.000,B 0.000,C 90.000,E1 47.391} C_DIS
LIN {X -0.332,Y -602.194,Z 1471.056,A 0.000,B 0.000,C 90.000,E1 46.134} C_DIS
LIN {X -0.091,Y -602.110,Z 1471.052,A 0.000,B 0.000,C 90.000,E1 45.324} C_DIS
LIN {X -0.259,Y -601.590,Z 1471.045,A 0.000,B 0.000,C 90.000,E1 44.028} C_DIS
LIN {X -0.005,Y -600.765,Z 1471.037,A 0.000,B 0.000,C 90.000,E1 42.690} C_DIS
LIN {X 0.043,Y -599.829,Z 1471.031,A 0.000,B 0.000,C 90.000,E1 41.634} C_DIS
LIN {X -0.369,Y -598.689,Z 1471.026,A 0.000,B 0.000,C 90.000,E1 40.620} C_DIS
LIN {X 0.112,Y -597.384,Z 1471.020,A 0.000,B 0.000,C 90.000,E1 39.519} C_DIS
LIN {X 0.112,Y -595.816,Z 1471.014,A 0.000,B 0.000,C 90.000,E1 38.463} C_DIS
LIN {X -0.286,Y -594.173,Z 1471.008,A 0.000,B 0.000,C 90.000,E1 37.443} C_DIS
LIN {X -0.016,Y -591.719,Z 1471.000,A 0.000,B 0.000,C 90.000,E1 36.091} C_DIS
LIN {X 0.001,Y -589.294,Z 1470.995,A 0.000,B 0.000,C 90.000,E1 35.025} C_DIS
LIN {X 0.070,Y -587.917,Z 1470.992,A 0.000,B 0.000,C 90.000,E1 34.485} C_DIS
LIN {X -0.161,Y -585.675,Z 1470.987,A 0.000,B 0.000,C 90.000,E1 33.706} C_DIS
LIN {X 0.067,Y -583.233,Z 1470.983,A 0.000,B 0.000,C 90.000,E1 32.880} C_DIS
LIN {X -0.044,Y -580.479,Z 1470.978,A 0.000,B 0.000,C 90.000,E1 32.084} C_DIS
LIN {X -0.028,Y -578.484,Z 1470.975,A 0.000,B 0.000,C 90.000,E1 31.544} C_DIS
LIN {X 0.115,Y -575.051,Z 1470.971,A 0.000,B 0.000,C 90.000,E1 30.718} C_DIS
LIN {X -0.201,Y -572.581,Z 1470.968,A 0.000,B 0.000,C 90.000,E1 30.207} C_DIS
LIN {X -0.163,Y -570.589,Z 1470.965,A 0.000,B 0.000,C 90.000,E1 29.795} C_DIS
LIN {X 0.001,Y -565.642,Z 1470.960,A 0.000,B 0.000,C 90.000,E1 28.821} C_DIS
LIN {X 0.202,Y -560.899,Z 1470.956,A 0.000,B 0.000,C 90.000,E1 27.975} C_DIS
LIN {X -0.196,Y -557.542,Z 1470.953,A 0.000,B 0.000,C 90.000,E1 27.462} C_DIS
LIN {X 0.241,Y -554.879,Z 1470.950,A 0.000,B 0.000,C 90.000,E1 27.001} C_DIS
LIN {X 0.071,Y -549.202,Z 1470.946,A 0.000,B 0.000,C 90.000,E1 26.181} C_DIS
LIN {X -0.043,Y -542.003,Z 1470.940,A 0.000,B 0.000,C 90.000,E1 25.207} C_DIS
LIN {X 0.146,Y -535.252,Z 1470.935,A 0.000,B 0.000,C 90.000,E1 24.335} C_DIS
LIN {X 0.070,Y -530.362,Z 1470.932,A 0.000,B 0.000,C 90.000,E1 23.770} C_DIS
LIN {X 0.206,Y -526.190,Z 1470.930,A 0.000,B 0.000,C 90.000,E1 23.334} C_DIS
LIN {X 0.164,Y -523.038,Z 1470.928,A 0.000,B 0.000,C 90.000,E1 23.078} C_DIS
LIN {X 0.132,Y -519.645,Z 1470.927,A 0.000,B 0.000,C 90.000,E1 22.845} C_DIS
LIN {X 0.056,Y -516.455,Z 1470.926,A 0.000,B 0.000,C 90.000,E1 22.695} C_DIS
LIN {X -0.032,Y -514.234,Z 1470.926,A 0.000,B 0.000,C 90.000,E1 22.642} C_DIS
LIN {X -0.064,Y -513.949,Z 1470.926,A 0.000,B 0.000,C 90.000,E1 22.642} C_DIS
LIN {X -0.072,Y -379.411,Z 1470.926,A 0.000,B 0.000,C 90.000,E1 22.642} C_DIS
LIN {X 0.073,Y -373.605,Z 1470.897,A 0.000,B 0.000,C 90.000,E1 17.457} C_DIS
LIN {X 0.107,Y -368.011,Z 1470.869,A 0.000,B 0.000,C 90.000,E1 12.299} C_DIS
LIN {X 0.124,Y -366.573,Z 1470.856,A 0.000,B 0.000,C 90.000,E1 10.074} C_DIS
LIN {X -0.020,Y -366.298,Z 1470.854,A 0.000,B 0.000,C 90.000,E1 9.726} C_DIS
LIN {X -0.141,Y -361.700,Z 1470.821,A 0.000,B 0.000,C 90.000,E1 3.784} C_DIS
LIN {X -0.060,Y -360.908,Z 1470.802,A 0.000,B 0.000,C 90.000,E1 0.401} C_DIS
LIN {X 0.137,Y -360.684,Z 1470.799,A 0.000,B 0.000,C 90.000,E1 359.771} C_DIS
LIN {X -0.053,Y -359.426,Z 1470.770,A 0.000,B 0.000,C 90.000,E1 354.546} C_DIS
LIN {X 0.070,Y -358.890,Z 1470.759,A 0.000,B 0.000,C 90.000,E1 352.648} C_DIS
LIN {X -0.020,Y -359.563,Z 1470.726,A 0.000,B 0.000,C 90.000,E1 346.645} C_DIS
LIN {X 0.001,Y -361.801,Z 1470.684,A 0.000,B 0.000,C 90.000,E1 339.135} C_DIS
LIN {X -0.154,Y -362.053,Z 1470.680,A 0.000,B 0.000,C 90.000,E1 338.411} C_DIS
LIN {X 0.189,Y -365.980,Z 1470.643,A 0.000,B 0.000,C 90.000,E1 331.641} C_DIS
LIN {X 0.029,Y -366.387,Z 1470.639,A 0.000,B 0.000,C 90.000,E1 330.923} C_DIS
LIN {X -0.031,Y -371.355,Z 1470.604,A 0.000,B 0.000,C 90.000,E1 324.642} C_DIS
LIN {X -0.043,Y -371.766,Z 1470.602,A 0.000,B 0.000,C 90.000,E1 324.276} C_DIS
LIN {X 0.013,Y -377.358,Z 1470.567,A 0.000,B 0.000,C 90.000,E1 318.038} C_DIS
LIN {X 0.012,Y -378.235,Z 1470.563,A 0.000,B 0.000,C 90.000,E1 317.310} C_DIS
LIN {X 0.002,Y -383.940,Z 1470.531,A 0.000,B 0.000,C 90.000,E1 311.515} C_DIS
LIN {X 0.088,Y -384.893,Z 1470.527,A 0.000,B 0.000,C 90.000,E1 310.782} C_DIS
LIN {X 0.262,Y -390.610,Z 1470.495,A 0.000,B 0.000,C 90.000,E1 305.025} C_DIS
LIN {X 0.106,Y -391.104,Z 1470.493,A 0.000,B 0.000,C 90.000,E1 304.692} C_DIS
LIN {X 0.022,Y -391.648,Z 1470.489,A 0.000,B 0.000,C 90.000,E1 303.992} C_DIS
LIN {X -0.080,Y -396.825,Z 1470.459,A 0.000,B 0.000,C 90.000,E1 298.693} C_DIS
LIN {X -0.210,Y -397.120,Z 1470.457,A 0.000,B 0.000,C 90.000,E1 298.359} C_DIS
LIN {X -0.055,Y -401.597,Z 1470.426,A 0.000,B 0.000,C 90.000,E1 292.717} C_DIS
LIN {X 0.222,Y -404.659,Z 1470.395,A 0.000,B 0.000,C 90.000,E1 287.094} C_DIS
LIN {X -0.079,Y -404.735,Z 1470.391,A 0.000,B 0.000,C 90.000,E1 286.441} C_DIS
LIN {X 0.214,Y -406.099,Z 1470.364,A 0.000,B 0.000,C 90.000,E1 281.535} C_DIS
LIN {X -0.176,Y -406.094,Z 1470.362,A 0.000,B 0.000,C 90.000,E1 281.243} C_DIS
LIN {X -0.097,Y -405.680,Z 1470.333,A 0.000,B 0.000,C 90.000,E1 276.024} C_DIS
LIN {X -0.165,Y -405.058,Z 1470.328,A 0.000,B 0.000,C 90.000,E1 274.992} C_DIS
LIN {X -0.060,Y -403.497,Z 1470.304,A 0.000,B 0.000,C 90.000,E1 270.802} C_DIS
LIN {X -0.092,Y -403.288,Z 1470.302,A 0.000,B 0.000,C 90.000,E1 270.458} C_DIS
LIN {X 0.091,Y -398.931,Z 1470.271,A 0.000,B 0.000,C 90.000,E1 264.837} C_DIS
LIN {X -0.040,Y -393.108,Z 1470.242,A 0.000,B 0.000,C 90.000,E1 259.567} C_DIS
LIN {X -0.079,Y -392.835,Z 1470.240,A 0.000,B 0.000,C 90.000,E1 259.218} C_DIS
LIN {X 0.034,Y -385.993,Z 1470.212,A 0.000,B 0.000,C 90.000,E1 254.212} C_DIS
LIN {X -0.026,Y -385.267,Z 1470.208,A 0.000,B 0.000,C 90.000,E1 253.504} C_DIS
LIN {X -0.004,Y -384.768,Z 1470.206,A 0.000,B 0.000,C 90.000,E1 253.142} C_DIS
LIN {X 0.221,Y -377.973,Z 1470.182,A 0.000,B 0.000,C 90.000,E1 248.773} C_DIS
LIN {X -0.044,Y -376.233,Z 1470.174,A 0.000,B 0.000,C 90.000,E1 247.358} C_DIS
LIN {X 0.057,Y -374.944,Z 1470.170,A 0.000,B 0.000,C 90.000,E1 246.613} C_DIS
LIN {X -0.208,Y -368.417,Z 1470.148,A 0.000,B 0.000,C 90.000,E1 242.615} C_DIS
LIN {X 0.097,Y -366.047,Z 1470.137,A 0.000,B 0.000,C 90.000,E1 240.717} C_DIS
LIN {X 0.004,Y -359.196,Z 1470.115,A 0.000,B 0.000,C 90.000,E1 236.628} C_DIS
LIN {X 0.021,Y -355.842,Z 1470.100,A 0.000,B 0.000,C 90.000,E1 233.989} C_DIS
LIN {X -0.173,Y -348.793,Z 1470.075,A 0.000,B 0.000,C 90.000,E1 229.461} C_DIS
LIN {X -0.097,Y -346.185,Z 1470.062,A 0.000,B 0.000,C 90.000,E1 227.148} C_DIS
LIN {X -0.088,Y -345.065,Z 1470.058,A 0.000,B 0.000,C 90.000,E1 226.377} C_DIS
LIN {X 0.094,Y -338.586,Z 1470.030,A 0.000,B 0.000,C 90.000,E1 221.310} C_DIS
LIN {X 0.094,Y -336.840,Z 1470.019,A 0.000,B 0.000,C 90.000,E1 219.358} C_DIS
LIN {X 0.014,Y -330.861,Z 1469.988,A 0.000,B 0.000,C 90.000,E1 213.865} C_DIS
LIN {X 0.149,Y -329.296,Z 1469.975,A 0.000,B 0.000,C 90.000,E1 211.465} C_DIS
LIN {X -0.154,Y -324.669,Z 1469.942,A 0.000,B 0.000,C 90.000,E1 205.540} C_DIS
LIN {X 0.174,Y -323.837,Z 1469.928,A 0.000,B 0.000,C 90.000,E1 203.078} C_DIS
LIN {X -0.017,Y -321.124,Z 1469.881,A 0.000,B 0.000,C 90.000,E1 194.662} C_DIS
LIN {X 0.138,Y -320.932,Z 1469.877,A 0.000,B 0.000,C 90.000,E1 193.828} C_DIS
LIN {X -0.076,Y -321.562,Z 1469.832,A 0.000,B 0.000,C 90.000,E1 185.796} C_DIS
LIN {X -0.143,Y -324.415,Z 1469.790,A 0.000,B 0.000,C 90.000,E1 178.165} C_DIS
LIN {X -0.141,Y -325.376,Z 1469.783,A 0.000,B 0.000,C 90.000,E1 176.963} C_DIS
LIN {X -0.100,Y -329.112,Z 1469.750,A 0.000,B 0.000,C 90.000,E1 170.971} C_DIS
LIN {X 0.061,Y -334.260,Z 1469.726,A 0.000,B 0.000,C 90.000,E1 166.589} C_DIS
LIN {X 0.067,Y -335.488,Z 1469.719,A 0.000,B 0.000,C 90.000,E1 165.408} C_DIS
LIN {X 0.143,Y -340.932,Z 1469.695,A 0.000,B 0.000,C 90.000,E1 161.094} C_DIS
LIN {X -0.172,Y -342.138,Z 1469.691,A 0.000,B 0.000,C 90.000,E1 160.369} C_DIS
LIN {X -0.147,Y -348.469,Z 1469.665,A 0.000,B 0.000,C 90.000,E1 155.793} C_DIS
LIN {X 0.185,Y -472.053,Z 1469.665,A 0.000,B 0.000,C 90.000,E1 155.741} C_DIS
LIN {X -0.078,Y -474.618,Z 1469.665,A 0.000,B 0.000,C 90.000,E1 155.717} C_DIS
LIN {X 0.086,Y -476.809,Z 1469.665,A 0.000,B 0.000,C 90.000,E1 155.613} C_DIS
LIN {X 0.020,Y -479.545,Z 1469.664,A 0.000,B 0.000,C 90.000,E1 155.485} C_DIS
LIN {X 0.110,Y -482.458,Z 1469.663,A 0.000,B 0.000,C 90.000,E1 155.305} C_DIS
LIN {X -0.068,Y -486.796,Z 1469.661,A 0.000,B 0.000,C 90.000,E1 155.025} C_DIS
LIN {X -0.015,Y -489.629,Z 1469.660,A 0.000,B 0.000,C 90.000,E1 154.793} C_DIS
LIN {X 0.070,Y -493.788,Z 1469.658,A 0.000,B 0.000,C 90.000,E1 154.409} C_DIS
LIN {X 0.153,Y -500.628,Z 1469.654,A 0.000,B 0.000,C 90.000,E1 153.717} C_DIS
LIN {X -0.128,Y -505.799,Z 1469.651,A 0.000,B 0.000,C 90.000,E1 153.179} C_DIS
LIN {X -0.176,Y -509.561,Z 1469.649,A 0.000,B 0.000,C 90.000,E1 152.743} C_DIS
LIN {X -0.209,Y -514.164,Z 1469.645,A 0.000,B 0.000,C 90.000,E1 152.153} C_DIS
LIN {X 0.251,Y -518.257,Z 1469.642,A 0.000,B 0.000,C 90.000,E1 151.513} C_DIS
LIN {X 0.288,Y -521.902,Z 1469.639,A 0.000,B 0.000,C 90.000,E1 150.923} C_DIS
LIN {X 0.193,Y -525.878,Z 1469.635,A 0.000,B 0.000,C 90.000,E1 150.205} C_DIS
LIN {X 0.128,Y -529.441,Z 1469.631,A 0.000,B 0.000,C 90.000,E1 149.488} C_DIS
LIN {X 0.061,Y -531.949,Z 1469.627,A 0.000,B 0.000,C 90.000,E1 148.918} C_DIS
LIN {X 0.195,Y -534.257,Z 1469.624,A 0.000,B 0.000,C 90.000,E1 148.329} C_DIS
LIN {X -0.120,Y -537.299,Z 1469.619,A 0.000,B 0.000,C 90.000,E1 147.502} C_DIS
LIN {X 0.052,Y -540.040,Z 1469.615,A 0.000,B 0.000,C 90.000,E1 146.628} C_DIS
LIN {X -0.200,Y -542.514,Z 1469.610,A 0.000,B 0.000,C 90.000,E1 145.801} C_DIS
LIN {X 0.328,Y -544.763,Z 1469.605,A 0.000,B 0.000,C 90.000,E1 144.895} C_DIS
LIN {X 0.120,Y -546.750,Z 1469.600,A 0.000,B 0.000,C 90.000,E1 144.069} C_DIS
LIN {X 0.250,Y -548.523,Z 1469.596,A 0.000,B 0.000,C 90.000,E1 143.210} C_DIS
LIN {X 0.021,Y -550.594,Z 1469.590,A 0.000,B 0.000,C 90.000,E1 142.110} C_DIS
LIN {X 0.194,Y -551.905,Z 1469.585,A 0.000,B 0.000,C 90.000,E1 141.251} C_DIS
LIN {X 0.010,Y -553.427,Z 1469.579,A 0.000,B 0.000,C 90.000,E1 140.150} C_DIS
